      "I171.4" { ExternalVisible := 'False'} : Bool := FALSE;   // I171.4
      "I171.5" { ExternalVisible := 'False'} : Bool := FALSE;   // I171.5
      "I171.6" { ExternalVisible := 'False'} : Bool := FALSE;   // I171.6
      "I171.7" { ExternalVisible := 'False'} : Bool := FALSE;   // I171.7
      "I172.0" { ExternalVisible := 'False'} : Bool := FALSE;   // I172.0
      "I172.1" { ExternalVisible := 'False'} : Bool := FALSE;   // I172.1
      "I172.2" { ExternalVisible := 'False'} : Bool := FALSE;   // I172.2
      "I172.3" { ExternalVisible := 'False'} : Bool := FALSE;   // I172.3
      "I172.4" { ExternalVisible := 'False'} : Bool := FALSE;   // I172.4
      "I172.5" { ExternalVisible := 'False'} : Bool := FALSE;   // I172.5
      "I172.6" { ExternalVisible := 'False'} : Bool := FALSE;   // I172.6
      "I172.7" { ExternalVisible := 'False'} : Bool := FALSE;   // I172.7
      "I173.0" { ExternalVisible := 'False'} : Bool := FALSE;   // I173.0
      "I173.1" { ExternalVisible := 'False'} : Bool := FALSE;   // I173.1
      "I173.2" { ExternalVisible := 'False'} : Bool := FALSE;   // I173.2
      "I173.3" { ExternalVisible := 'False'} : Bool := FALSE;   // I173.3
      "I173.4" { ExternalVisible := 'False'} : Bool := FALSE;   // I173.4
      "I173.5" { ExternalVisible := 'False'} : Bool := FALSE;   // I173.5
      "I173.6" { ExternalVisible := 'False'} : Bool := FALSE;   // I173.6
      "I173.7" { ExternalVisible := 'False'} : Bool := FALSE;   // I173.7
      "I174.0" { ExternalVisible := 'False'} : Bool := FALSE;   // I174.0
      "I174.1" { ExternalVisible := 'False'} : Bool := FALSE;   // I174.1
      "I174.2" { ExternalVisible := 'False'} : Bool := FALSE;   // I174.2
      "I174.3" { ExternalVisible := 'False'} : Bool := FALSE;   // I174.3
      "I174.4" { ExternalVisible := 'False'} : Bool := FALSE;   // I174.4
      "I174.5" { ExternalVisible := 'False'} : Bool := FALSE;   // I174.5
      "I174.6" { ExternalVisible := 'False'} : Bool := FALSE;   // I174.6
      "I174.7" { ExternalVisible := 'False'} : Bool := FALSE;   // I174.7
      "I175.0" { ExternalVisible := 'False'} : Bool := FALSE;   // I175.0
      "I175.1" { ExternalVisible := 'False'} : Bool := FALSE;   // I175.1
      "I175.2" { ExternalVisible := 'False'} : Bool := FALSE;   // I175.2
      "I175.3" { ExternalVisible := 'False'} : Bool := FALSE;   // I175.3
      "I175.4" { ExternalVisible := 'False'} : Bool := FALSE;   // I175.4
      "I175.5" { ExternalVisible := 'False'} : Bool := FALSE;   // I175.5
      "I175.6" { ExternalVisible := 'False'} : Bool := FALSE;   // I175.6
      "I175.7" { ExternalVisible := 'False'} : Bool := FALSE;   // I175.7
      "I176.0" { ExternalVisible := 'False'} : Bool := FALSE;   // I176.0
      "I176.1" { ExternalVisible := 'False'} : Bool := FALSE;   // I176.1
      "I176.2" { ExternalVisible := 'False'} : Bool := FALSE;   // I176.2
      "I176.3" { ExternalVisible := 'False'} : Bool := FALSE;   // I176.3
      "I176.4" { ExternalVisible := 'False'} : Bool := FALSE;   // I176.4
      "I176.5" { ExternalVisible := 'False'} : Bool := FALSE;   // I176.5
      "I176.6" { ExternalVisible := 'False'} : Bool := FALSE;   // I176.6
      "I176.7" { ExternalVisible := 'False'} : Bool := FALSE;   // I176.7
      "I177.0" { ExternalVisible := 'False'} : Bool := FALSE;   // I177.0
      "I177.1" { ExternalVisible := 'False'} : Bool := FALSE;   // I177.1
      "I177.2" { ExternalVisible := 'False'} : Bool := FALSE;   // I177.2
      "I177.3" { ExternalVisible := 'False'} : Bool := FALSE;   // I177.3
      "I177.4" { ExternalVisible := 'False'} : Bool := FALSE;   // I177.4
      "I177.5" { ExternalVisible := 'False'} : Bool := FALSE;   // I177.5
      "I177.6" { ExternalVisible := 'False'} : Bool := FALSE;   // I177.6
      "I177.7" { ExternalVisible := 'False'} : Bool := FALSE;   // I177.7
      "I178.0" { ExternalVisible := 'False'} : Bool := FALSE;   // I178.0
      "I178.1" { ExternalVisible := 'False'} : Bool := FALSE;   // I178.1
      "I178.2" { ExternalVisible := 'False'} : Bool := FALSE;   // I178.2
      "I178.3" { ExternalVisible := 'False'} : Bool := FALSE;   // I178.3
      "I178.4" { ExternalVisible := 'False'} : Bool := FALSE;   // I178.4
      "I178.5" { ExternalVisible := 'False'} : Bool := FALSE;   // I178.5
      "I178.6" { ExternalVisible := 'False'} : Bool := FALSE;   // I178.6
      "I178.7" { ExternalVisible := 'False'} : Bool := FALSE;   // I178.7
      "I179.0" { ExternalVisible := 'False'} : Bool := FALSE;   // I179.0
      "I179.1" { ExternalVisible := 'False'} : Bool := FALSE;   // I179.1
      "I179.2" { ExternalVisible := 'False'} : Bool := FALSE;   // I179.2
      "I179.3" { ExternalVisible := 'False'} : Bool := FALSE;   // I179.3
      "I179.4" { ExternalVisible := 'False'} : Bool := FALSE;   // I179.4
      "I179.5" { ExternalVisible := 'False'} : Bool := FALSE;   // I179.5
      "I179.6" { ExternalVisible := 'False'} : Bool := FALSE;   // I179.6
      "I179.7" { ExternalVisible := 'False'} : Bool := FALSE;   // I179.7
      "I180.0" { ExternalVisible := 'False'} : Bool := FALSE;   // I180.0
      "I180.1" { ExternalVisible := 'False'} : Bool := FALSE;   // I180.1
      "I180.2" { ExternalVisible := 'False'} : Bool := FALSE;   // I180.2
      "I180.3" { ExternalVisible := 'False'} : Bool := FALSE;   // I180.3
      "I180.4" { ExternalVisible := 'False'} : Bool := FALSE;   // I180.4
      "I180.5" { ExternalVisible := 'False'} : Bool := FALSE;   // I180.5
      "I180.6" { ExternalVisible := 'False'} : Bool := FALSE;   // I180.6
      "I180.7" { ExternalVisible := 'False'} : Bool := FALSE;   // I180.7
      "I181.0" { ExternalVisible := 'False'} : Bool := FALSE;   // I181.0
      "I181.1" { ExternalVisible := 'False'} : Bool := FALSE;   // I181.1
      "I181.2" { ExternalVisible := 'False'} : Bool := FALSE;   // I181.2
      "I181.3" { ExternalVisible := 'False'} : Bool := FALSE;   // I181.3
      "I181.4" { ExternalVisible := 'False'} : Bool := FALSE;   // I181.4
      "I181.5" { ExternalVisible := 'False'} : Bool := FALSE;   // I181.5
      "I181.6" { ExternalVisible := 'False'} : Bool := FALSE;   // I181.6
      "I181.7" { ExternalVisible := 'False'} : Bool := FALSE;   // I181.7
      "I182.0" { ExternalVisible := 'False'} : Bool := FALSE;   // I182.0
      "I182.1" { ExternalVisible := 'False'} : Bool := FALSE;   // I182.1
      "I182.2" { ExternalVisible := 'False'} : Bool := FALSE;   // I182.2
      "I182.3" { ExternalVisible := 'False'} : Bool := FALSE;   // I182.3
      "I182.4" { ExternalVisible := 'False'} : Bool := FALSE;   // I182.4
      "I182.5" { ExternalVisible := 'False'} : Bool := FALSE;   // I182.5
      "I182.6" { ExternalVisible := 'False'} : Bool := FALSE;   // I182.6
      "I182.7" { ExternalVisible := 'False'} : Bool := FALSE;   // I182.7
      "I183.0" { ExternalVisible := 'False'} : Bool := FALSE;   // I183.0
      "I183.1" { ExternalVisible := 'False'} : Bool := FALSE;   // I183.1
      "I183.2" { ExternalVisible := 'False'} : Bool := FALSE;   // I183.2
      "I183.3" { ExternalVisible := 'False'} : Bool := FALSE;   // I183.3
      "I183.4" { ExternalVisible := 'False'} : Bool := FALSE;   // I183.4
      "I183.5" { ExternalVisible := 'False'} : Bool := FALSE;   // I183.5
      "I183.6" { ExternalVisible := 'False'} : Bool := FALSE;   // I183.6
      "I183.7" { ExternalVisible := 'False'} : Bool := FALSE;   // I183.7
      "I184.0" { ExternalVisible := 'False'} : Bool := FALSE;   // I184.0
      "I184.1" { ExternalVisible := 'False'} : Bool := FALSE;   // I184.1
      "I184.2" { ExternalVisible := 'False'} : Bool := FALSE;   // I184.2
      "I184.3" { ExternalVisible := 'False'} : Bool := FALSE;   // I184.3
      "I184.4" { ExternalVisible := 'False'} : Bool := FALSE;   // I184.4
      "I184.5" { ExternalVisible := 'False'} : Bool := FALSE;   // I184.5
      "I184.6" { ExternalVisible := 'False'} : Bool := FALSE;   // I184.6
      "I184.7" { ExternalVisible := 'False'} : Bool := FALSE;   // I184.7
      "I185.0" { ExternalVisible := 'False'} : Bool := FALSE;   // I185.0
      "I185.1" { ExternalVisible := 'False'} : Bool := FALSE;   // I185.1
      "I185.2" { ExternalVisible := 'False'} : Bool := FALSE;   // I185.2
      "I185.3" { ExternalVisible := 'False'} : Bool := FALSE;   // I185.3
      "I185.4" { ExternalVisible := 'False'} : Bool := FALSE;   // I185.4
      "I185.5" { ExternalVisible := 'False'} : Bool := FALSE;   // I185.5
      "I185.6" { ExternalVisible := 'False'} : Bool := FALSE;   // I185.6
      "I185.7" { ExternalVisible := 'False'} : Bool := FALSE;   // I185.7
      "I186.0" { ExternalVisible := 'False'} : Bool := FALSE;   // I186.0
      "I186.1" { ExternalVisible := 'False'} : Bool := FALSE;   // I186.1
      "I186.2" { ExternalVisible := 'False'} : Bool := FALSE;   // I186.2
      "I186.3" { ExternalVisible := 'False'} : Bool := FALSE;   // I186.3
      "I186.4" { ExternalVisible := 'False'} : Bool := FALSE;   // I186.4
      "I186.5" { ExternalVisible := 'False'} : Bool := FALSE;   // I186.5
      "I186.6" { ExternalVisible := 'False'} : Bool := FALSE;   // I186.6
      "I186.7" { ExternalVisible := 'False'} : Bool := FALSE;   // I186.7
      "I187.0" { ExternalVisible := 'False'} : Bool := FALSE;   // I187.0
      "I187.1" { ExternalVisible := 'False'} : Bool := FALSE;   // I187.1
      "I187.2" { ExternalVisible := 'False'} : Bool := FALSE;   // I187.2
      "I187.3" { ExternalVisible := 'False'} : Bool := FALSE;   // I187.3
      "I187.4" { ExternalVisible := 'False'} : Bool := FALSE;   // I187.4
      "I187.5" { ExternalVisible := 'False'} : Bool := FALSE;   // I187.5
      "I187.6" { ExternalVisible := 'False'} : Bool := FALSE;   // I187.6
      "I187.7" { ExternalVisible := 'False'} : Bool := FALSE;   // I187.7
      "I188.0" { ExternalVisible := 'False'} : Bool := FALSE;   // I188.0
      "I188.1" { ExternalVisible := 'False'} : Bool := FALSE;   // I188.1
      "I188.2" { ExternalVisible := 'False'} : Bool := FALSE;   // I188.2
      "I188.3" { ExternalVisible := 'False'} : Bool := FALSE;   // I188.3
      "I188.4" { ExternalVisible := 'False'} : Bool := FALSE;   // I188.4
      "I188.5" { ExternalVisible := 'False'} : Bool := FALSE;   // I188.5
      "I188.6" { ExternalVisible := 'False'} : Bool := FALSE;   // I188.6
      "I188.7" { ExternalVisible := 'False'} : Bool := FALSE;   // I188.7
      "I189.0" { ExternalVisible := 'False'} : Bool := FALSE;   // I189.0
      "I189.1" { ExternalVisible := 'False'} : Bool := FALSE;   // I189.1
      "I189.2" { ExternalVisible := 'False'} : Bool := FALSE;   // I189.2
      "I189.3" { ExternalVisible := 'False'} : Bool := FALSE;   // I189.3
      "I189.4" { ExternalVisible := 'False'} : Bool := FALSE;   // I189.4
      "I189.5" { ExternalVisible := 'False'} : Bool := FALSE;   // I189.5
      "I189.6" { ExternalVisible := 'False'} : Bool := FALSE;   // I189.6
      "I189.7" { ExternalVisible := 'False'} : Bool := FALSE;   // I189.7
      "I190.0" { ExternalVisible := 'False'} : Bool := FALSE;   // I190.0
      "I190.1" { ExternalVisible := 'False'} : Bool := FALSE;   // I190.1
      "I190.2" { ExternalVisible := 'False'} : Bool := FALSE;   // I190.2
      "I190.3" { ExternalVisible := 'False'} : Bool := FALSE;   // I190.3
      "I190.4" { ExternalVisible := 'False'} : Bool := FALSE;   // I190.4
      "I190.5" { ExternalVisible := 'False'} : Bool := FALSE;   // I190.5
      "I190.6" { ExternalVisible := 'False'} : Bool := FALSE;   // I190.6
      "I190.7" { ExternalVisible := 'False'} : Bool := FALSE;   // I190.7
      "I191.0" { ExternalVisible := 'False'} : Bool := FALSE;   // I191.0
      "I191.1" { ExternalVisible := 'False'} : Bool := FALSE;   // I191.1
      "I191.2" { ExternalVisible := 'False'} : Bool := FALSE;   // I191.2
      "I191.3" { ExternalVisible := 'False'} : Bool := FALSE;   // I191.3
      "I191.4" { ExternalVisible := 'False'} : Bool := FALSE;   // I191.4
      "I191.5" { ExternalVisible := 'False'} : Bool := FALSE;   // I191.5
      "I191.6" { ExternalVisible := 'False'} : Bool := FALSE;   // I191.6
      "I191.7" { ExternalVisible := 'False'} : Bool := FALSE;   // I191.7
      "I192.0" { ExternalVisible := 'False'} : Bool := FALSE;   // I192.0
      "I192.1" { ExternalVisible := 'False'} : Bool := FALSE;   // I192.1
      "I192.2" { ExternalVisible := 'False'} : Bool := FALSE;   // I192.2
      "I192.3" { ExternalVisible := 'False'} : Bool := FALSE;   // I192.3
      "I192.4" { ExternalVisible := 'False'} : Bool := FALSE;   // I192.4
      "I192.5" { ExternalVisible := 'False'} : Bool := FALSE;   // I192.5
      "I192.6" { ExternalVisible := 'False'} : Bool := FALSE;   // I192.6
      "I192.7" { ExternalVisible := 'False'} : Bool := FALSE;   // I192.7
      "I193.0" { ExternalVisible := 'False'} : Bool := FALSE;   // I193.0
      "I193.1" { ExternalVisible := 'False'} : Bool := FALSE;   // I193.1
      "I193.2" { ExternalVisible := 'False'} : Bool := FALSE;   // I193.2
      "I193.3" { ExternalVisible := 'False'} : Bool := FALSE;   // I193.3
      "I193.4" { ExternalVisible := 'False'} : Bool := FALSE;   // I193.4
      "I193.5" { ExternalVisible := 'False'} : Bool := FALSE;   // I193.5
      "I193.6" { ExternalVisible := 'False'} : Bool := FALSE;   // I193.6
      "I193.7" { ExternalVisible := 'False'} : Bool := FALSE;   // I193.7
      "I194.0" { ExternalVisible := 'False'} : Bool := FALSE;   // I194.0
      "I194.1" { ExternalVisible := 'False'} : Bool := FALSE;   // I194.1
      "I194.2" { ExternalVisible := 'False'} : Bool := FALSE;   // I194.2
      "I194.3" { ExternalVisible := 'False'} : Bool := FALSE;   // I194.3
      "I194.4" { ExternalVisible := 'False'} : Bool := FALSE;   // I194.4
      "I194.5" { ExternalVisible := 'False'} : Bool := FALSE;   // I194.5
      "I194.6" { ExternalVisible := 'False'} : Bool := FALSE;   // I194.6
      "I194.7" { ExternalVisible := 'False'} : Bool := FALSE;   // I194.7
      "I195.0" { ExternalVisible := 'False'} : Bool := FALSE;   // I195.0
      "I195.1" { ExternalVisible := 'False'} : Bool := FALSE;   // I195.1
      "I195.2" { ExternalVisible := 'False'} : Bool := FALSE;   // I195.2
      "I195.3" { ExternalVisible := 'False'} : Bool := FALSE;   // I195.3
      "I195.4" { ExternalVisible := 'False'} : Bool := FALSE;   // I195.4
      "I195.5" { ExternalVisible := 'False'} : Bool := FALSE;   // I195.5
      "I195.6" { ExternalVisible := 'False'} : Bool := FALSE;   // I195.6
      "I195.7" { ExternalVisible := 'False'} : Bool := FALSE;   // I195.7
      "I196.0" { ExternalVisible := 'False'} : Bool := FALSE;   // I196.0
      "I196.1" { ExternalVisible := 'False'} : Bool := FALSE;   // I196.1
      "I196.2" { ExternalVisible := 'False'} : Bool := FALSE;   // I196.2
      "I196.3" { ExternalVisible := 'False'} : Bool := FALSE;   // I196.3
      "I196.4" { ExternalVisible := 'False'} : Bool := FALSE;   // I196.4
      "I196.5" { ExternalVisible := 'False'} : Bool := FALSE;   // I196.5
      "I196.6" { ExternalVisible := 'False'} : Bool := FALSE;   // I196.6
      "I196.7" { ExternalVisible := 'False'} : Bool := FALSE;   // I196.7
      "I197.0" { ExternalVisible := 'False'} : Bool := FALSE;   // I197.0
      "I197.1" { ExternalVisible := 'False'} : Bool := FALSE;   // I197.1
      "I197.2" { ExternalVisible := 'False'} : Bool := FALSE;   // I197.2
      "I197.3" { ExternalVisible := 'False'} : Bool := FALSE;   // I197.3
      "I197.4" { ExternalVisible := 'False'} : Bool := FALSE;   // I197.4
      "I197.5" { ExternalVisible := 'False'} : Bool := FALSE;   // I197.5
      "I197.6" { ExternalVisible := 'False'} : Bool := FALSE;   // I197.6
      "I197.7" { ExternalVisible := 'False'} : Bool := FALSE;   // I197.7
      "I198.0" { ExternalVisible := 'False'} : Bool := FALSE;   // I198.0
      "I198.1" { ExternalVisible := 'False'} : Bool := FALSE;   // I198.1
      "I198.2" { ExternalVisible := 'False'} : Bool := FALSE;   // I198.2
      "I198.3" { ExternalVisible := 'False'} : Bool := FALSE;   // I198.3
      "I198.4" { ExternalVisible := 'False'} : Bool := FALSE;   // I198.4
      "I198.5" { ExternalVisible := 'False'} : Bool := FALSE;   // I198.5
      "I198.6" { ExternalVisible := 'False'} : Bool := FALSE;   // I198.6
      "I198.7" { ExternalVisible := 'False'} : Bool := FALSE;   // I198.7
      "I199.0" { ExternalVisible := 'False'} : Bool := FALSE;   // I199.0
      "I199.1" { ExternalVisible := 'False'} : Bool := FALSE;   // I199.1
      "I199.2" { ExternalVisible := 'False'} : Bool := FALSE;   // I199.2
      "I199.3" { ExternalVisible := 'False'} : Bool := FALSE;   // I199.3
      "I199.4" { ExternalVisible := 'False'} : Bool := FALSE;   // I199.4
      "I199.5" { ExternalVisible := 'False'} : Bool := FALSE;   // I199.5
      "I199.6" { ExternalVisible := 'False'} : Bool := FALSE;   // I199.6
      "I199.7" { ExternalVisible := 'False'} : Bool := FALSE;   // I199.7
      "I200.0" { ExternalVisible := 'False'} : Bool := FALSE;   // I200.0
      "I200.1" { ExternalVisible := 'False'} : Bool := FALSE;   // I200.1
      "I200.2" { ExternalVisible := 'False'} : Bool := FALSE;   // I200.2
      "I200.3" { ExternalVisible := 'False'} : Bool := FALSE;   // I200.3
      "I200.4" { ExternalVisible := 'False'} : Bool := FALSE;   // I200.4
      "I200.5" { ExternalVisible := 'False'} : Bool := FALSE;   // I200.5
      "I200.6" { ExternalVisible := 'False'} : Bool := FALSE;   // I200.6
      "I200.7" { ExternalVisible := 'False'} : Bool := FALSE;   // I200.7
      "I201.0" { ExternalVisible := 'False'} : Bool := FALSE;   // I201.0
      "I201.1" { ExternalVisible := 'False'} : Bool := FALSE;   // I201.1
      "I201.2" { ExternalVisible := 'False'} : Bool := FALSE;   // I201.2
      "I201.3" { ExternalVisible := 'False'} : Bool := FALSE;   // I201.3
      "I201.4" { ExternalVisible := 'False'} : Bool := FALSE;   // I201.4
      "I201.5" { ExternalVisible := 'False'} : Bool := FALSE;   // I201.5
      "I201.6" { ExternalVisible := 'False'} : Bool := FALSE;   // I201.6
      "I201.7" { ExternalVisible := 'False'} : Bool := FALSE;   // I201.7
      "I202.0" { ExternalVisible := 'False'} : Bool := FALSE;   // I202.0
      "I202.1" { ExternalVisible := 'False'} : Bool := FALSE;   // I202.1
      "I202.2" { ExternalVisible := 'False'} : Bool := FALSE;   // I202.2
      "I202.3" { ExternalVisible := 'False'} : Bool := FALSE;   // I202.3
      "I202.4" { ExternalVisible := 'False'} : Bool := FALSE;   // I202.4
      "I202.5" { ExternalVisible := 'False'} : Bool := FALSE;   // I202.5
      "I202.6" { ExternalVisible := 'False'} : Bool := FALSE;   // I202.6
      "I202.7" { ExternalVisible := 'False'} : Bool := FALSE;   // I202.7
      "I203.0" { ExternalVisible := 'False'} : Bool := FALSE;   // I203.0
      "I203.1" { ExternalVisible := 'False'} : Bool := FALSE;   // I203.1
      "I203.2" { ExternalVisible := 'False'} : Bool := FALSE;   // I203.2
      "I203.3" { ExternalVisible := 'False'} : Bool := FALSE;   // I203.3
      "I203.4" { ExternalVisible := 'False'} : Bool := FALSE;   // I203.4
      "I203.5" { ExternalVisible := 'False'} : Bool := FALSE;   // I203.5
      "I203.6" { ExternalVisible := 'False'} : Bool := FALSE;   // I203.6
      "I203.7" { ExternalVisible := 'False'} : Bool := FALSE;   // I203.7
      "I204.0" { ExternalVisible := 'False'} : Bool := FALSE;   // I204.0
      "I204.1" { ExternalVisible := 'False'} : Bool := FALSE;   // I204.1
      "I204.2" { ExternalVisible := 'False'} : Bool := FALSE;   // I204.2
      "I204.3" { ExternalVisible := 'False'} : Bool := FALSE;   // I204.3
      "I204.4" { ExternalVisible := 'False'} : Bool := FALSE;   // I204.4
      "I204.5" { ExternalVisible := 'False'} : Bool := FALSE;   // I204.5
      "I204.6" { ExternalVisible := 'False'} : Bool := FALSE;   // I204.6
      "I204.7" { ExternalVisible := 'False'} : Bool := FALSE;   // I204.7
      "I205.0" { ExternalVisible := 'False'} : Bool := FALSE;   // I205.0
      "I205.1" { ExternalVisible := 'False'} : Bool := FALSE;   // I205.1
      "I205.2" { ExternalVisible := 'False'} : Bool := FALSE;   // I205.2
      "I205.3" { ExternalVisible := 'False'} : Bool := FALSE;   // I205.3
      "I205.4" { ExternalVisible := 'False'} : Bool := FALSE;   // I205.4
      "I205.5" { ExternalVisible := 'False'} : Bool := FALSE;   // I205.5
      "I205.6" { ExternalVisible := 'False'} : Bool := FALSE;   // I205.6
      "I205.7" { ExternalVisible := 'False'} : Bool := FALSE;   // I205.7
      "I206.0" { ExternalVisible := 'False'} : Bool := FALSE;   // I206.0
      "I206.1" { ExternalVisible := 'False'} : Bool := FALSE;   // I206.1
      "I206.2" { ExternalVisible := 'False'} : Bool := FALSE;   // I206.2
      "I206.3" { ExternalVisible := 'False'} : Bool := FALSE;   // I206.3
      "I206.4" { ExternalVisible := 'False'} : Bool := FALSE;   // I206.4
      "I206.5" { ExternalVisible := 'False'} : Bool := FALSE;   // I206.5
      "I206.6" { ExternalVisible := 'False'} : Bool := FALSE;   // I206.6
      "I206.7" { ExternalVisible := 'False'} : Bool := FALSE;   // I206.7
      "I207.0" { ExternalVisible := 'False'} : Bool := FALSE;   // I207.0
      "I207.1" { ExternalVisible := 'False'} : Bool := FALSE;   // I207.1
      "I207.2" { ExternalVisible := 'False'} : Bool := FALSE;   // I207.2
      "I207.3" { ExternalVisible := 'False'} : Bool := FALSE;   // I207.3
      "I207.4" { ExternalVisible := 'False'} : Bool := FALSE;   // I207.4
      "I207.5" { ExternalVisible := 'False'} : Bool := FALSE;   // I207.5
      "I207.6" { ExternalVisible := 'False'} : Bool := FALSE;   // I207.6
      "I207.7" { ExternalVisible := 'False'} : Bool := FALSE;   // I207.7
      "I208.0" { ExternalVisible := 'False'} : Bool := FALSE;   // I208.0
      "I208.1" { ExternalVisible := 'False'} : Bool := FALSE;   // I208.1
      "I208.2" { ExternalVisible := 'False'} : Bool := FALSE;   // I208.2
      "I208.3" { ExternalVisible := 'False'} : Bool := FALSE;   // I208.3
      "I208.4" { ExternalVisible := 'False'} : Bool := FALSE;   // I208.4
      "I208.5" { ExternalVisible := 'False'} : Bool := FALSE;   // I208.5
      "I208.6" { ExternalVisible := 'False'} : Bool := FALSE;   // I208.6
      "I208.7" { ExternalVisible := 'False'} : Bool := FALSE;   // I208.7
      "I209.0" { ExternalVisible := 'False'} : Bool := FALSE;   // I209.0
      "I209.1" { ExternalVisible := 'False'} : Bool := FALSE;   // I209.1
      "I209.2" { ExternalVisible := 'False'} : Bool := FALSE;   // I209.2
      "I209.3" { ExternalVisible := 'False'} : Bool := FALSE;   // I209.3
      "I209.4" { ExternalVisible := 'False'} : Bool := FALSE;   // I209.4
      "I209.5" { ExternalVisible := 'False'} : Bool := FALSE;   // I209.5
      "I209.6" { ExternalVisible := 'False'} : Bool := FALSE;   // I209.6
      "I209.7" { ExternalVisible := 'False'} : Bool := FALSE;   // I209.7
      "I210.0" { ExternalVisible := 'False'} : Bool := FALSE;   // I210.0
      "I210.1" { ExternalVisible := 'False'} : Bool := FALSE;   // I210.1
      "I210.2" { ExternalVisible := 'False'} : Bool := FALSE;   // I210.2
      "I210.3" { ExternalVisible := 'False'} : Bool := FALSE;   // I210.3
      "I210.4" { ExternalVisible := 'False'} : Bool := FALSE;   // I210.4
      "I210.5" { ExternalVisible := 'False'} : Bool := FALSE;   // I210.5
      "I210.6" { ExternalVisible := 'False'} : Bool := FALSE;   // I210.6
      "I210.7" { ExternalVisible := 'False'} : Bool := FALSE;   // I210.7
      "I211.0" { ExternalVisible := 'False'} : Bool := FALSE;   // I211.0
      "I211.1" { ExternalVisible := 'False'} : Bool := FALSE;   // I211.1
      "I211.2" { ExternalVisible := 'False'} : Bool := FALSE;   // I211.2
      "I211.3" { ExternalVisible := 'False'} : Bool := FALSE;   // I211.3
      "I211.4" { ExternalVisible := 'False'} : Bool := FALSE;   // I211.4
      "I211.5" { ExternalVisible := 'False'} : Bool := FALSE;   // I211.5
      "I211.6" { ExternalVisible := 'False'} : Bool := FALSE;   // I211.6
      "I211.7" { ExternalVisible := 'False'} : Bool := FALSE;   // I211.7
      "I212.0" { ExternalVisible := 'False'} : Bool := FALSE;   // I212.0
      "I212.1" { ExternalVisible := 'False'} : Bool := FALSE;   // I212.1
      "I212.2" { ExternalVisible := 'False'} : Bool := FALSE;   // I212.2
      "I212.3" { ExternalVisible := 'False'} : Bool := FALSE;   // I212.3
      "I212.4" { ExternalVisible := 'False'} : Bool := FALSE;   // I212.4
      "I212.5" { ExternalVisible := 'False'} : Bool := FALSE;   // I212.5
      "I212.6" { ExternalVisible := 'False'} : Bool := FALSE;   // I212.6
      "I212.7" { ExternalVisible := 'False'} : Bool := FALSE;   // I212.7
      "I213.0" { ExternalVisible := 'False'} : Bool := FALSE;   // I213.0
      "I213.1" { ExternalVisible := 'False'} : Bool := FALSE;   // I213.1
      "I213.2" { ExternalVisible := 'False'} : Bool := FALSE;   // I213.2
      "I213.3" { ExternalVisible := 'False'} : Bool := FALSE;   // I213.3
      "I213.4" { ExternalVisible := 'False'} : Bool := FALSE;   // I213.4
      "I213.5" { ExternalVisible := 'False'} : Bool := FALSE;   // I213.5
      "I213.6" { ExternalVisible := 'False'} : Bool := FALSE;   // I213.6
      "I213.7" { ExternalVisible := 'False'} : Bool := FALSE;   // I213.7
      "I214.0" { ExternalVisible := 'False'} : Bool := FALSE;   // I214.0
      "I214.1" { ExternalVisible := 'False'} : Bool := FALSE;   // I214.1
      "I214.2" { ExternalVisible := 'False'} : Bool := FALSE;   // I214.2
      "I214.3" { ExternalVisible := 'False'} : Bool := FALSE;   // I214.3
      "I214.4" { ExternalVisible := 'False'} : Bool := FALSE;   // I214.4
      "I214.5" { ExternalVisible := 'False'} : Bool := FALSE;   // I214.5
      "I214.6" { ExternalVisible := 'False'} : Bool := FALSE;   // I214.6
      "I214.7" { ExternalVisible := 'False'} : Bool := FALSE;   // I214.7
      "I215.0" { ExternalVisible := 'False'} : Bool := FALSE;   // I215.0
      "I215.1" { ExternalVisible := 'False'} : Bool := FALSE;   // I215.1
      "I215.2" { ExternalVisible := 'False'} : Bool := FALSE;   // I215.2
      "I215.3" { ExternalVisible := 'False'} : Bool := FALSE;   // I215.3
      "I215.4" { ExternalVisible := 'False'} : Bool := FALSE;   // I215.4
      "I215.5" { ExternalVisible := 'False'} : Bool := FALSE;   // I215.5
      "I215.6" { ExternalVisible := 'False'} : Bool := FALSE;   // I215.6
      "I215.7" { ExternalVisible := 'False'} : Bool := FALSE;   // I215.7
      "I216.0" { ExternalVisible := 'False'} : Bool := FALSE;   // I216.0
      "I216.1" { ExternalVisible := 'False'} : Bool := FALSE;   // I216.1
      "I216.2" { ExternalVisible := 'False'} : Bool := FALSE;   // I216.2
      "I216.3" { ExternalVisible := 'False'} : Bool := FALSE;   // I216.3
      "I216.4" { ExternalVisible := 'False'} : Bool := FALSE;   // I216.4
      "I216.5" { ExternalVisible := 'False'} : Bool := FALSE;   // I216.5
      "I216.6" { ExternalVisible := 'False'} : Bool := FALSE;   // I216.6
      "I216.7" { ExternalVisible := 'False'} : Bool := FALSE;   // I216.7
      "I217.0" { ExternalVisible := 'False'} : Bool := FALSE;   // I217.0
      "I217.1" { ExternalVisible := 'False'} : Bool := FALSE;   // I217.1
      "I217.2" { ExternalVisible := 'False'} : Bool := FALSE;   // I217.2
      "I217.3" { ExternalVisible := 'False'} : Bool := FALSE;   // I217.3
      "I217.4" { ExternalVisible := 'False'} : Bool := FALSE;   // I217.4
      "I217.5" { ExternalVisible := 'False'} : Bool := FALSE;   // I217.5
      "I217.6" { ExternalVisible := 'False'} : Bool := FALSE;   // I217.6
      "I217.7" { ExternalVisible := 'False'} : Bool := FALSE;   // I217.7
      "I218.0" { ExternalVisible := 'False'} : Bool := FALSE;   // I218.0
      "I218.1" { ExternalVisible := 'False'} : Bool := FALSE;   // I218.1
      "I218.2" { ExternalVisible := 'False'} : Bool := FALSE;   // I218.2
      "I218.3" { ExternalVisible := 'False'} : Bool := FALSE;   // I218.3
      "I218.4" { ExternalVisible := 'False'} : Bool := FALSE;   // I218.4
      "I218.5" { ExternalVisible := 'False'} : Bool := FALSE;   // I218.5
      "I218.6" { ExternalVisible := 'False'} : Bool := FALSE;   // I218.6
      "I218.7" { ExternalVisible := 'False'} : Bool := FALSE;   // I218.7
      "I219.0" { ExternalVisible := 'False'} : Bool := FALSE;   // I219.0
      "I219.1" { ExternalVisible := 'False'} : Bool := FALSE;   // I219.1
      "I219.2" { ExternalVisible := 'False'} : Bool := FALSE;   // I219.2
      "I219.3" { ExternalVisible := 'False'} : Bool := FALSE;   // I219.3
      "I219.4" { ExternalVisible := 'False'} : Bool := FALSE;   // I219.4
      "I219.5" { ExternalVisible := 'False'} : Bool := FALSE;   // I219.5
      "I219.6" { ExternalVisible := 'False'} : Bool := FALSE;   // I219.6
      "I219.7" { ExternalVisible := 'False'} : Bool := FALSE;   // I219.7
      "I220.0" { ExternalVisible := 'False'} : Bool := FALSE;   // I220.0
      "I220.1" { ExternalVisible := 'False'} : Bool := FALSE;   // I220.1
      "I220.2" { ExternalVisible := 'False'} : Bool := FALSE;   // I220.2
      "I220.3" { ExternalVisible := 'False'} : Bool := FALSE;   // I220.3
      "I220.4" { ExternalVisible := 'False'} : Bool := FALSE;   // I220.4
      "I220.5" { ExternalVisible := 'False'} : Bool := FALSE;   // I220.5
      "I220.6" { ExternalVisible := 'False'} : Bool := FALSE;   // I220.6
      "I220.7" { ExternalVisible := 'False'} : Bool := FALSE;   // I220.7
      "I221.0" { ExternalVisible := 'False'} : Bool := FALSE;   // I221.0
      "I221.1" { ExternalVisible := 'False'} : Bool := FALSE;   // I221.1
      "I221.2" { ExternalVisible := 'False'} : Bool := FALSE;   // I221.2
      "I221.3" { ExternalVisible := 'False'} : Bool := FALSE;   // I221.3
      "I221.4" { ExternalVisible := 'False'} : Bool := FALSE;   // I221.4
      "I221.5" { ExternalVisible := 'False'} : Bool := FALSE;   // I221.5
      "I221.6" { ExternalVisible := 'False'} : Bool := FALSE;   // I221.6
      "I221.7" { ExternalVisible := 'False'} : Bool := FALSE;   // I221.7
      "I222.0" { ExternalVisible := 'False'} : Bool := FALSE;   // I222.0
      "I222.1" { ExternalVisible := 'False'} : Bool := FALSE;   // I222.1
      "I222.2" { ExternalVisible := 'False'} : Bool := FALSE;   // I222.2
      "I222.3" { ExternalVisible := 'False'} : Bool := FALSE;   // I222.3
      "I222.4" { ExternalVisible := 'False'} : Bool := FALSE;   // I222.4
      "I222.5" { ExternalVisible := 'False'} : Bool := FALSE;   // I222.5
      "I222.6" { ExternalVisible := 'False'} : Bool := FALSE;   // I222.6
      "I222.7" { ExternalVisible := 'False'} : Bool := FALSE;   // I222.7
      "I223.0" { ExternalVisible := 'False'} : Bool := FALSE;   // I223.0
      "I223.1" { ExternalVisible := 'False'} : Bool := FALSE;   // I223.1
      "I223.2" { ExternalVisible := 'False'} : Bool := FALSE;   // I223.2
      "I223.3" { ExternalVisible := 'False'} : Bool := FALSE;   // I223.3
      "I223.4" { ExternalVisible := 'False'} : Bool := FALSE;   // I223.4
      "I223.5" { ExternalVisible := 'False'} : Bool := FALSE;   // I223.5
      "I223.6" { ExternalVisible := 'False'} : Bool := FALSE;   // I223.6
      "I223.7" { ExternalVisible := 'False'} : Bool := FALSE;   // I223.7
      "I224.0" { ExternalVisible := 'False'} : Bool := FALSE;   // I224.0
      "I224.1" { ExternalVisible := 'False'} : Bool := FALSE;   // I224.1
      "I224.2" { ExternalVisible := 'False'} : Bool := FALSE;   // I224.2
      "I224.3" { ExternalVisible := 'False'} : Bool := FALSE;   // I224.3
      "I224.4" { ExternalVisible := 'False'} : Bool := FALSE;   // I224.4
      "I224.5" { ExternalVisible := 'False'} : Bool := FALSE;   // I224.5
      "I224.6" { ExternalVisible := 'False'} : Bool := FALSE;   // I224.6
      "I224.7" { ExternalVisible := 'False'} : Bool := FALSE;   // I224.7
      "I225.0" { ExternalVisible := 'False'} : Bool := FALSE;   // I225.0
      "I225.1" { ExternalVisible := 'False'} : Bool := FALSE;   // I225.1
      "I225.2" { ExternalVisible := 'False'} : Bool := FALSE;   // I225.2
      "I225.3" { ExternalVisible := 'False'} : Bool := FALSE;   // I225.3
      "I225.4" { ExternalVisible := 'False'} : Bool := FALSE;   // I225.4
      "I225.5" { ExternalVisible := 'False'} : Bool := FALSE;   // I225.5
      "I225.6" { ExternalVisible := 'False'} : Bool := FALSE;   // I225.6
      "I225.7" { ExternalVisible := 'False'} : Bool := FALSE;   // I225.7
      "I226.0" { ExternalVisible := 'False'} : Bool := FALSE;   // I226.0
      "I226.1" { ExternalVisible := 'False'} : Bool := FALSE;   // I226.1
      "I226.2" { ExternalVisible := 'False'} : Bool := FALSE;   // I226.2
      "I226.3" { ExternalVisible := 'False'} : Bool := FALSE;   // I226.3
      "I226.4" { ExternalVisible := 'False'} : Bool := FALSE;   // I226.4
      "I226.5" { ExternalVisible := 'False'} : Bool := FALSE;   // I226.5
      "I226.6" { ExternalVisible := 'False'} : Bool := FALSE;   // I226.6
      "I226.7" { ExternalVisible := 'False'} : Bool := FALSE;   // I226.7
      "I227.0" { ExternalVisible := 'False'} : Bool := FALSE;   // I227.0
      "I227.1" { ExternalVisible := 'False'} : Bool := FALSE;   // I227.1
      "I227.2" { ExternalVisible := 'False'} : Bool := FALSE;   // I227.2
      "I227.3" { ExternalVisible := 'False'} : Bool := FALSE;   // I227.3
      "I227.4" { ExternalVisible := 'False'} : Bool := FALSE;   // I227.4
      "I227.5" { ExternalVisible := 'False'} : Bool := FALSE;   // I227.5
      "I227.6" { ExternalVisible := 'False'} : Bool := FALSE;   // I227.6
      "I227.7" { ExternalVisible := 'False'} : Bool := FALSE;   // I227.7
      "I228.0" { ExternalVisible := 'False'} : Bool := FALSE;   // I228.0
      "I228.1" { ExternalVisible := 'False'} : Bool := FALSE;   // I228.1
      "I228.2" { ExternalVisible := 'False'} : Bool := FALSE;   // I228.2
      "I228.3" { ExternalVisible := 'False'} : Bool := FALSE;   // I228.3
      "I228.4" { ExternalVisible := 'False'} : Bool := FALSE;   // I228.4
      "I228.5" { ExternalVisible := 'False'} : Bool := FALSE;   // I228.5
      "I228.6" { ExternalVisible := 'False'} : Bool := FALSE;   // I228.6
      "I228.7" { ExternalVisible := 'False'} : Bool := FALSE;   // I228.7
      "I229.0" { ExternalVisible := 'False'} : Bool := FALSE;   // I229.0
      "I229.1" { ExternalVisible := 'False'} : Bool := FALSE;   // I229.1
      "I229.2" { ExternalVisible := 'False'} : Bool := FALSE;   // I229.2
      "I229.3" { ExternalVisible := 'False'} : Bool := FALSE;   // I229.3
      "I229.4" { ExternalVisible := 'False'} : Bool := FALSE;   // I229.4
      "I229.5" { ExternalVisible := 'False'} : Bool := FALSE;   // I229.5
      "I229.6" { ExternalVisible := 'False'} : Bool := FALSE;   // I229.6
      "I229.7" { ExternalVisible := 'False'} : Bool := FALSE;   // I229.7
      "I230.0" { ExternalVisible := 'False'} : Bool := FALSE;   // I230.0
      "I230.1" { ExternalVisible := 'False'} : Bool := FALSE;   // I230.1
      "I230.2" { ExternalVisible := 'False'} : Bool := FALSE;   // I230.2
      "I230.3" { ExternalVisible := 'False'} : Bool := FALSE;   // I230.3
      "I230.4" { ExternalVisible := 'False'} : Bool := FALSE;   // I230.4
      "I230.5" { ExternalVisible := 'False'} : Bool := FALSE;   // I230.5
      "I230.6" { ExternalVisible := 'False'} : Bool := FALSE;   // I230.6
      "I230.7" { ExternalVisible := 'False'} : Bool := FALSE;   // I230.7
      "I231.0" { ExternalVisible := 'False'} : Bool := FALSE;   // I231.0
      "I231.1" { ExternalVisible := 'False'} : Bool := FALSE;   // I231.1
      "I231.2" { ExternalVisible := 'False'} : Bool := FALSE;   // I231.2
      "I231.3" { ExternalVisible := 'False'} : Bool := FALSE;   // I231.3
      "I231.4" { ExternalVisible := 'False'} : Bool := FALSE;   // I231.4
      "I231.5" { ExternalVisible := 'False'} : Bool := FALSE;   // I231.5
      "I231.6" { ExternalVisible := 'False'} : Bool := FALSE;   // I231.6
      "I231.7" { ExternalVisible := 'False'} : Bool := FALSE;   // I231.7
      "I232.0" { ExternalVisible := 'False'} : Bool := FALSE;   // I232.0
      "I232.1" { ExternalVisible := 'False'} : Bool := FALSE;   // I232.1
      "I232.2" { ExternalVisible := 'False'} : Bool := FALSE;   // I232.2
      "I232.3" { ExternalVisible := 'False'} : Bool := FALSE;   // I232.3
      "I232.4" { ExternalVisible := 'False'} : Bool := FALSE;   // I232.4
      "I232.5" { ExternalVisible := 'False'} : Bool := FALSE;   // I232.5
      "I232.6" { ExternalVisible := 'False'} : Bool := FALSE;   // I232.6
      "I232.7" { ExternalVisible := 'False'} : Bool := FALSE;   // I232.7
      "I233.0" { ExternalVisible := 'False'} : Bool := FALSE;   // I233.0
      "I233.1" { ExternalVisible := 'False'} : Bool := FALSE;   // I233.1
      "I233.2" { ExternalVisible := 'False'} : Bool := FALSE;   // I233.2
      "I233.3" { ExternalVisible := 'False'} : Bool := FALSE;   // I233.3
      "I233.4" { ExternalVisible := 'False'} : Bool := FALSE;   // I233.4
      "I233.5" { ExternalVisible := 'False'} : Bool := FALSE;   // I233.5
      "I233.6" { ExternalVisible := 'False'} : Bool := FALSE;   // I233.6
      "I233.7" { ExternalVisible := 'False'} : Bool := FALSE;   // I233.7
      "I234.0" { ExternalVisible := 'False'} : Bool := FALSE;   // I234.0
      "I234.1" { ExternalVisible := 'False'} : Bool := FALSE;   // I234.1
      "I234.2" { ExternalVisible := 'False'} : Bool := FALSE;   // I234.2
      "I234.3" { ExternalVisible := 'False'} : Bool := FALSE;   // I234.3
      "I234.4" { ExternalVisible := 'False'} : Bool := FALSE;   // I234.4
      "I234.5" { ExternalVisible := 'False'} : Bool := FALSE;   // I234.5
      "I234.6" { ExternalVisible := 'False'} : Bool := FALSE;   // I234.6
      "I234.7" { ExternalVisible := 'False'} : Bool := FALSE;   // I234.7
      "I235.0" { ExternalVisible := 'False'} : Bool := FALSE;   // I235.0
      "I235.1" { ExternalVisible := 'False'} : Bool := FALSE;   // I235.1
      "I235.2" { ExternalVisible := 'False'} : Bool := FALSE;   // I235.2
      "I235.3" { ExternalVisible := 'False'} : Bool := FALSE;   // I235.3
      "I235.4" { ExternalVisible := 'False'} : Bool := FALSE;   // I235.4
      "I235.5" { ExternalVisible := 'False'} : Bool := FALSE;   // I235.5
      "I235.6" { ExternalVisible := 'False'} : Bool := FALSE;   // I235.6
      "I235.7" { ExternalVisible := 'False'} : Bool := FALSE;   // I235.7
      "I236.0" { ExternalVisible := 'False'} : Bool := FALSE;   // I236.0
      "I236.1" { ExternalVisible := 'False'} : Bool := FALSE;   // I236.1
      "I236.2" { ExternalVisible := 'False'} : Bool := FALSE;   // I236.2
      "I236.3" { ExternalVisible := 'False'} : Bool := FALSE;   // I236.3
      "I236.4" { ExternalVisible := 'False'} : Bool := FALSE;   // I236.4
      "I236.5" { ExternalVisible := 'False'} : Bool := FALSE;   // I236.5
      "I236.6" { ExternalVisible := 'False'} : Bool := FALSE;   // I236.6
      "I236.7" { ExternalVisible := 'False'} : Bool := FALSE;   // I236.7
      "I237.0" { ExternalVisible := 'False'} : Bool := FALSE;   // I237.0
      "I237.1" { ExternalVisible := 'False'} : Bool := FALSE;   // I237.1
      "I237.2" { ExternalVisible := 'False'} : Bool := FALSE;   // I237.2
      "I237.3" { ExternalVisible := 'False'} : Bool := FALSE;   // I237.3
      "I237.4" { ExternalVisible := 'False'} : Bool := FALSE;   // I237.4
      "I237.5" { ExternalVisible := 'False'} : Bool := FALSE;   // I237.5
      "I237.6" { ExternalVisible := 'False'} : Bool := FALSE;   // I237.6
      "I237.7" { ExternalVisible := 'False'} : Bool := FALSE;   // I237.7
      "I238.0" { ExternalVisible := 'False'} : Bool := FALSE;   // I238.0
      "I238.1" { ExternalVisible := 'False'} : Bool := FALSE;   // I238.1
      "I238.2" { ExternalVisible := 'False'} : Bool := FALSE;   // I238.2
      "I238.3" { ExternalVisible := 'False'} : Bool := FALSE;   // I238.3
      "I238.4" { ExternalVisible := 'False'} : Bool := FALSE;   // I238.4
      "I238.5" { ExternalVisible := 'False'} : Bool := FALSE;   // I238.5
      "I238.6" { ExternalVisible := 'False'} : Bool := FALSE;   // I238.6
      "I238.7" { ExternalVisible := 'False'} : Bool := FALSE;   // I238.7
      "I239.0" { ExternalVisible := 'False'} : Bool := FALSE;   // I239.0
      "I239.1" { ExternalVisible := 'False'} : Bool := FALSE;   // I239.1
      "I239.2" { ExternalVisible := 'False'} : Bool := FALSE;   // I239.2
      "I239.3" { ExternalVisible := 'False'} : Bool := FALSE;   // I239.3
      "I239.4" { ExternalVisible := 'False'} : Bool := FALSE;   // I239.4
      "I239.5" { ExternalVisible := 'False'} : Bool := FALSE;   // I239.5
      "I239.6" { ExternalVisible := 'False'} : Bool := FALSE;   // I239.6
      "I239.7" { ExternalVisible := 'False'} : Bool := FALSE;   // I239.7
      "I240.0" { ExternalVisible := 'False'} : Bool := FALSE;   // I240.0
      "I240.1" { ExternalVisible := 'False'} : Bool := FALSE;   // I240.1
      "I240.2" { ExternalVisible := 'False'} : Bool := FALSE;   // I240.2
      "I240.3" { ExternalVisible := 'False'} : Bool := FALSE;   // I240.3
      "I240.4" { ExternalVisible := 'False'} : Bool := FALSE;   // I240.4
      "I240.5" { ExternalVisible := 'False'} : Bool := FALSE;   // I240.5
      "I240.6" { ExternalVisible := 'False'} : Bool := FALSE;   // I240.6
      "I240.7" { ExternalVisible := 'False'} : Bool := FALSE;   // I240.7
      "I241.0" { ExternalVisible := 'False'} : Bool := FALSE;   // I241.0
      "I241.1" { ExternalVisible := 'False'} : Bool := FALSE;   // I241.1
      "I241.2" { ExternalVisible := 'False'} : Bool := FALSE;   // I241.2
      "I241.3" { ExternalVisible := 'False'} : Bool := FALSE;   // I241.3
      "I241.4" { ExternalVisible := 'False'} : Bool := FALSE;   // I241.4
      "I241.5" { ExternalVisible := 'False'} : Bool := FALSE;   // I241.5
      "I241.6" { ExternalVisible := 'False'} : Bool := FALSE;   // I241.6
      "I241.7" { ExternalVisible := 'False'} : Bool := FALSE;   // I241.7
      "I242.0" { ExternalVisible := 'False'} : Bool := FALSE;   // I242.0
      "I242.1" { ExternalVisible := 'False'} : Bool := FALSE;   // I242.1
      "I242.2" { ExternalVisible := 'False'} : Bool := FALSE;   // I242.2
      "I242.3" { ExternalVisible := 'False'} : Bool := FALSE;   // I242.3
      "I242.4" { ExternalVisible := 'False'} : Bool := FALSE;   // I242.4
      "I242.5" { ExternalVisible := 'False'} : Bool := FALSE;   // I242.5
      "I242.6" { ExternalVisible := 'False'} : Bool := FALSE;   // I242.6
      "I242.7" { ExternalVisible := 'False'} : Bool := FALSE;   // I242.7
      "I243.0" { ExternalVisible := 'False'} : Bool := FALSE;   // I243.0
      "I243.1" { ExternalVisible := 'False'} : Bool := FALSE;   // I243.1
      "I243.2" { ExternalVisible := 'False'} : Bool := FALSE;   // I243.2
      "I243.3" { ExternalVisible := 'False'} : Bool := FALSE;   // I243.3
      "I243.4" { ExternalVisible := 'False'} : Bool := FALSE;   // I243.4
      "I243.5" { ExternalVisible := 'False'} : Bool := FALSE;   // I243.5
      "I243.6" { ExternalVisible := 'False'} : Bool := FALSE;   // I243.6
      "I243.7" { ExternalVisible := 'False'} : Bool := FALSE;   // I243.7
      "I244.0" { ExternalVisible := 'False'} : Bool := FALSE;   // I244.0
      "I244.1" { ExternalVisible := 'False'} : Bool := FALSE;   // I244.1
      "I244.2" { ExternalVisible := 'False'} : Bool := FALSE;   // I244.2
      "I244.3" { ExternalVisible := 'False'} : Bool := FALSE;   // I244.3
      "I244.4" { ExternalVisible := 'False'} : Bool := FALSE;   // I244.4
      "I244.5" { ExternalVisible := 'False'} : Bool := FALSE;   // I244.5
      "I244.6" { ExternalVisible := 'False'} : Bool := FALSE;   // I244.6
      "I244.7" { ExternalVisible := 'False'} : Bool := FALSE;   // I244.7
      "I245.0" { ExternalVisible := 'False'} : Bool := FALSE;   // I245.0
      "I245.1" { ExternalVisible := 'False'} : Bool := FALSE;   // I245.1
      "I245.2" { ExternalVisible := 'False'} : Bool := FALSE;   // I245.2
      "I245.3" { ExternalVisible := 'False'} : Bool := FALSE;   // I245.3
      "I245.4" { ExternalVisible := 'False'} : Bool := FALSE;   // I245.4
      "I245.5" { ExternalVisible := 'False'} : Bool := FALSE;   // I245.5
      "I245.6" { ExternalVisible := 'False'} : Bool := FALSE;   // I245.6
      "I245.7" { ExternalVisible := 'False'} : Bool := FALSE;   // I245.7
      "I246.0" { ExternalVisible := 'False'} : Bool := FALSE;   // I246.0
      "I246.1" { ExternalVisible := 'False'} : Bool := FALSE;   // I246.1
      "I246.2" { ExternalVisible := 'False'} : Bool := FALSE;   // I246.2
      "I246.3" { ExternalVisible := 'False'} : Bool := FALSE;   // I246.3
      "I246.4" { ExternalVisible := 'False'} : Bool := FALSE;   // I246.4
      "I246.5" { ExternalVisible := 'False'} : Bool := FALSE;   // I246.5
      "I246.6" { ExternalVisible := 'False'} : Bool := FALSE;   // I246.6
      "I246.7" { ExternalVisible := 'False'} : Bool := FALSE;   // I246.7
      "I247.0" { ExternalVisible := 'False'} : Bool := FALSE;   // I247.0
      "I247.1" { ExternalVisible := 'False'} : Bool := FALSE;   // I247.1
      "I247.2" { ExternalVisible := 'False'} : Bool := FALSE;   // I247.2
      "I247.3" { ExternalVisible := 'False'} : Bool := FALSE;   // I247.3
      "I247.4" { ExternalVisible := 'False'} : Bool := FALSE;   // I247.4
      "I247.5" { ExternalVisible := 'False'} : Bool := FALSE;   // I247.5
      "I247.6" { ExternalVisible := 'False'} : Bool := FALSE;   // I247.6
      "I247.7" { ExternalVisible := 'False'} : Bool := FALSE;   // I247.7
      "I248.0" { ExternalVisible := 'False'} : Bool := FALSE;   // I248.0
      "I248.1" { ExternalVisible := 'False'} : Bool := FALSE;   // I248.1
      "I248.2" { ExternalVisible := 'False'} : Bool := FALSE;   // I248.2
      "I248.3" { ExternalVisible := 'False'} : Bool := FALSE;   // I248.3
      "I248.4" { ExternalVisible := 'False'} : Bool := FALSE;   // I248.4
      "I248.5" { ExternalVisible := 'False'} : Bool := FALSE;   // I248.5
      "I248.6" { ExternalVisible := 'False'} : Bool := FALSE;   // I248.6
      "I248.7" { ExternalVisible := 'False'} : Bool := FALSE;   // I248.7
      "I249.0" { ExternalVisible := 'False'} : Bool := FALSE;   // I249.0
      "I249.1" { ExternalVisible := 'False'} : Bool := FALSE;   // I249.1
      "I249.2" { ExternalVisible := 'False'} : Bool := FALSE;   // I249.2
      "I249.3" { ExternalVisible := 'False'} : Bool := FALSE;   // I249.3
      "I249.4" { ExternalVisible := 'False'} : Bool := FALSE;   // I249.4
      "I249.5" { ExternalVisible := 'False'} : Bool := FALSE;   // I249.5
      "I249.6" { ExternalVisible := 'False'} : Bool := FALSE;   // I249.6
      "I249.7" { ExternalVisible := 'False'} : Bool := FALSE;   // I249.7
      "I250.0" { ExternalVisible := 'False'} : Bool := FALSE;   // I250.0
      "I250.1" { ExternalVisible := 'False'} : Bool := FALSE;   // I250.1
      "I250.2" { ExternalVisible := 'False'} : Bool := FALSE;   // I250.2
      "I250.3" { ExternalVisible := 'False'} : Bool := FALSE;   // I250.3
      "I250.4" { ExternalVisible := 'False'} : Bool := FALSE;   // I250.4
      "I250.5" { ExternalVisible := 'False'} : Bool := FALSE;   // I250.5
      "I250.6" { ExternalVisible := 'False'} : Bool := FALSE;   // I250.6
      "I250.7" { ExternalVisible := 'False'} : Bool := FALSE;   // I250.7
      "I251.0" { ExternalVisible := 'False'} : Bool := FALSE;   // I251.0
      "I251.1" { ExternalVisible := 'False'} : Bool := FALSE;   // I251.1
      "I251.2" { ExternalVisible := 'False'} : Bool := FALSE;   // I251.2
      "I251.3" { ExternalVisible := 'False'} : Bool := FALSE;   // I251.3
      "I251.4" { ExternalVisible := 'False'} : Bool := FALSE;   // I251.4
      "I251.5" { ExternalVisible := 'False'} : Bool := FALSE;   // I251.5
      "I251.6" { ExternalVisible := 'False'} : Bool := FALSE;   // I251.6
      "I251.7" { ExternalVisible := 'False'} : Bool := FALSE;   // I251.7
      "I252.0" { ExternalVisible := 'False'} : Bool := FALSE;   // I252.0
      "I252.1" { ExternalVisible := 'False'} : Bool := FALSE;   // I252.1
      "I252.2" { ExternalVisible := 'False'} : Bool := FALSE;   // I252.2
      "I252.3" { ExternalVisible := 'False'} : Bool := FALSE;   // I252.3
      "I252.4" { ExternalVisible := 'False'} : Bool := FALSE;   // I252.4
      "I252.5" { ExternalVisible := 'False'} : Bool := FALSE;   // I252.5
      "I252.6" { ExternalVisible := 'False'} : Bool := FALSE;   // I252.6
      "I252.7" { ExternalVisible := 'False'} : Bool := FALSE;   // I252.7
      "I253.0" { ExternalVisible := 'False'} : Bool := FALSE;   // I253.0
      "I253.1" { ExternalVisible := 'False'} : Bool := FALSE;   // I253.1
      "I253.2" { ExternalVisible := 'False'} : Bool := FALSE;   // I253.2
      "I253.3" { ExternalVisible := 'False'} : Bool := FALSE;   // I253.3
      "I253.4" { ExternalVisible := 'False'} : Bool := FALSE;   // I253.4
      "I253.5" { ExternalVisible := 'False'} : Bool := FALSE;   // I253.5
      "I253.6" { ExternalVisible := 'False'} : Bool := FALSE;   // I253.6
      "I253.7" { ExternalVisible := 'False'} : Bool := FALSE;   // I253.7
      "I254.0" { ExternalVisible := 'False'} : Bool := FALSE;   // I254.0
      "I254.1" { ExternalVisible := 'False'} : Bool := FALSE;   // I254.1
      "I254.2" { ExternalVisible := 'False'} : Bool := FALSE;   // I254.2
      "I254.3" { ExternalVisible := 'False'} : Bool := FALSE;   // I254.3
      "I254.4" { ExternalVisible := 'False'} : Bool := FALSE;   // I254.4
      "I254.5" { ExternalVisible := 'False'} : Bool := FALSE;   // I254.5
      "I254.6" { ExternalVisible := 'False'} : Bool := FALSE;   // I254.6
      "I254.7" { ExternalVisible := 'False'} : Bool := FALSE;   // I254.7
      "I255.0" { ExternalVisible := 'False'} : Bool := FALSE;   // I255.0
      "I255.1" { ExternalVisible := 'False'} : Bool := FALSE;   // I255.1
      "I255.2" { ExternalVisible := 'False'} : Bool := FALSE;   // I255.2
      "I255.3" { ExternalVisible := 'False'} : Bool := FALSE;   // I255.3
      "I255.4" { ExternalVisible := 'False'} : Bool := FALSE;   // I255.4
      "I255.5" { ExternalVisible := 'False'} : Bool := FALSE;   // I255.5
      "I255.6" { ExternalVisible := 'False'} : Bool := FALSE;   // I255.6
      "I255.7" { ExternalVisible := 'False'} : Bool := FALSE;   // I255.7
      "I256.0" { ExternalVisible := 'False'} : Bool := FALSE;   // I256.0
      "I256.1" { ExternalVisible := 'False'} : Bool := FALSE;   // I256.1
      "I256.2" { ExternalVisible := 'False'} : Bool := FALSE;   // I256.2
      "I256.3" { ExternalVisible := 'False'} : Bool := FALSE;   // I256.3
      "I256.4" { ExternalVisible := 'False'} : Bool := FALSE;   // I256.4
      "I256.5" { ExternalVisible := 'False'} : Bool := FALSE;   // I256.5
      "I256.6" { ExternalVisible := 'False'} : Bool := FALSE;   // I256.6
      "I256.7" { ExternalVisible := 'False'} : Bool := FALSE;   // I256.7
      "I257.0" { ExternalVisible := 'False'} : Bool := FALSE;   // I257.0
      "I257.1" { ExternalVisible := 'False'} : Bool := FALSE;   // I257.1
      "I257.2" { ExternalVisible := 'False'} : Bool := FALSE;   // I257.2
      "I257.3" { ExternalVisible := 'False'} : Bool := FALSE;   // I257.3
      "I257.4" { ExternalVisible := 'False'} : Bool := FALSE;   // I257.4
      "I257.5" { ExternalVisible := 'False'} : Bool := FALSE;   // I257.5
      "I257.6" { ExternalVisible := 'False'} : Bool := FALSE;   // I257.6
      "I257.7" { ExternalVisible := 'False'} : Bool := FALSE;   // I257.7
      "I258.0" { ExternalVisible := 'False'} : Bool := FALSE;   // I258.0
      "I258.1" { ExternalVisible := 'False'} : Bool := FALSE;   // I258.1
      "I258.2" { ExternalVisible := 'False'} : Bool := FALSE;   // I258.2
      "I258.3" { ExternalVisible := 'False'} : Bool := FALSE;   // I258.3
      "I258.4" { ExternalVisible := 'False'} : Bool := FALSE;   // I258.4
      "I258.5" { ExternalVisible := 'False'} : Bool := FALSE;   // I258.5
      "I258.6" { ExternalVisible := 'False'} : Bool := FALSE;   // I258.6
      "I258.7" { ExternalVisible := 'False'} : Bool := FALSE;   // I258.7
      "I259.0" { ExternalVisible := 'False'} : Bool := FALSE;   // I259.0
      "I259.1" { ExternalVisible := 'False'} : Bool := FALSE;   // I259.1
      "I259.2" { ExternalVisible := 'False'} : Bool := FALSE;   // I259.2
      "I259.3" { ExternalVisible := 'False'} : Bool := FALSE;   // I259.3
      "I259.4" { ExternalVisible := 'False'} : Bool := FALSE;   // I259.4
      "I259.5" { ExternalVisible := 'False'} : Bool := FALSE;   // I259.5
      "I259.6" { ExternalVisible := 'False'} : Bool := FALSE;   // I259.6
      "I259.7" { ExternalVisible := 'False'} : Bool := FALSE;   // I259.7
      "I260.0" { ExternalVisible := 'False'} : Bool := FALSE;   // I260.0
      "I260.1" { ExternalVisible := 'False'} : Bool := FALSE;   // I260.1
      "I260.2" { ExternalVisible := 'False'} : Bool := FALSE;   // I260.2
      "I260.3" { ExternalVisible := 'False'} : Bool := FALSE;   // I260.3
      "I260.4" { ExternalVisible := 'False'} : Bool := FALSE;   // I260.4
      "I260.5" { ExternalVisible := 'False'} : Bool := FALSE;   // I260.5
      "I260.6" { ExternalVisible := 'False'} : Bool := FALSE;   // I260.6
      "I260.7" { ExternalVisible := 'False'} : Bool := FALSE;   // I260.7
      "I261.0" { ExternalVisible := 'False'} : Bool := FALSE;   // I261.0
      "I261.1" { ExternalVisible := 'False'} : Bool := FALSE;   // I261.1
      "I261.2" { ExternalVisible := 'False'} : Bool := FALSE;   // I261.2
      "I261.3" { ExternalVisible := 'False'} : Bool := FALSE;   // I261.3
      "I261.4" { ExternalVisible := 'False'} : Bool := FALSE;   // I261.4
      "I261.5" { ExternalVisible := 'False'} : Bool := FALSE;   // I261.5
      "I261.6" { ExternalVisible := 'False'} : Bool := FALSE;   // I261.6
      "I261.7" { ExternalVisible := 'False'} : Bool := FALSE;   // I261.7
      "I262.0" { ExternalVisible := 'False'} : Bool := FALSE;   // I262.0
      "I262.1" { ExternalVisible := 'False'} : Bool := FALSE;   // I262.1
      "I262.2" { ExternalVisible := 'False'} : Bool := FALSE;   // I262.2
      "I262.3" { ExternalVisible := 'False'} : Bool := FALSE;   // I262.3
      "I262.4" { ExternalVisible := 'False'} : Bool := FALSE;   // I262.4
      "I262.5" { ExternalVisible := 'False'} : Bool := FALSE;   // I262.5
      "I262.6" { ExternalVisible := 'False'} : Bool := FALSE;   // I262.6
      "I262.7" { ExternalVisible := 'False'} : Bool := FALSE;   // I262.7
      "I263.0" { ExternalVisible := 'False'} : Bool := FALSE;   // I263.0
      "I263.1" { ExternalVisible := 'False'} : Bool := FALSE;   // I263.1
      "I263.2" { ExternalVisible := 'False'} : Bool := FALSE;   // I263.2
      "I263.3" { ExternalVisible := 'False'} : Bool := FALSE;   // I263.3
      "I263.4" { ExternalVisible := 'False'} : Bool := FALSE;   // I263.4
      "I263.5" { ExternalVisible := 'False'} : Bool := FALSE;   // I263.5
      "I263.6" { ExternalVisible := 'False'} : Bool := FALSE;   // I263.6
      "I263.7" { ExternalVisible := 'False'} : Bool := FALSE;   // I263.7
      "I264.0" { ExternalVisible := 'False'} : Bool := FALSE;   // I264.0
      "I264.1" { ExternalVisible := 'False'} : Bool := FALSE;   // I264.1
      "I264.2" { ExternalVisible := 'False'} : Bool := FALSE;   // I264.2
      "I264.3" { ExternalVisible := 'False'} : Bool := FALSE;   // I264.3
      "I264.4" { ExternalVisible := 'False'} : Bool := FALSE;   // I264.4
      "I264.5" { ExternalVisible := 'False'} : Bool := FALSE;   // I264.5
      "I264.6" { ExternalVisible := 'False'} : Bool := FALSE;   // I264.6
      "I264.7" { ExternalVisible := 'False'} : Bool := FALSE;   // I264.7
      "I265.0" { ExternalVisible := 'False'} : Bool := FALSE;   // I265.0
      "I265.1" { ExternalVisible := 'False'} : Bool := FALSE;   // I265.1
      "I265.2" { ExternalVisible := 'False'} : Bool := FALSE;   // I265.2
      "I265.3" { ExternalVisible := 'False'} : Bool := FALSE;   // I265.3
      "I265.4" { ExternalVisible := 'False'} : Bool := FALSE;   // I265.4
      "I265.5" { ExternalVisible := 'False'} : Bool := FALSE;   // I265.5
      "I265.6" { ExternalVisible := 'False'} : Bool := FALSE;   // I265.6
      "I265.7" { ExternalVisible := 'False'} : Bool := FALSE;   // I265.7
      "I266.0" { ExternalVisible := 'False'} : Bool := FALSE;   // I266.0
      "I266.1" { ExternalVisible := 'False'} : Bool := FALSE;   // I266.1
      "I266.2" { ExternalVisible := 'False'} : Bool := FALSE;   // I266.2
      "I266.3" { ExternalVisible := 'False'} : Bool := FALSE;   // I266.3
      "I266.4" { ExternalVisible := 'False'} : Bool := FALSE;   // I266.4
      "I266.5" { ExternalVisible := 'False'} : Bool := FALSE;   // I266.5
      "I266.6" { ExternalVisible := 'False'} : Bool := FALSE;   // I266.6
      "I266.7" { ExternalVisible := 'False'} : Bool := FALSE;   // I266.7
      "I267.0" { ExternalVisible := 'False'} : Bool := FALSE;   // I267.0
      "I267.1" { ExternalVisible := 'False'} : Bool := FALSE;   // I267.1
      "I267.2" { ExternalVisible := 'False'} : Bool := FALSE;   // I267.2
      "I267.3" { ExternalVisible := 'False'} : Bool := FALSE;   // I267.3
      "I267.4" { ExternalVisible := 'False'} : Bool := FALSE;   // I267.4
      "I267.5" { ExternalVisible := 'False'} : Bool := FALSE;   // I267.5
      "I267.6" { ExternalVisible := 'False'} : Bool := FALSE;   // I267.6
      "I267.7" { ExternalVisible := 'False'} : Bool := FALSE;   // I267.7
      "I268.0" { ExternalVisible := 'False'} : Bool := FALSE;   // I268.0
      "I268.1" { ExternalVisible := 'False'} : Bool := FALSE;   // I268.1
      "I268.2" { ExternalVisible := 'False'} : Bool := FALSE;   // I268.2
      "I268.3" { ExternalVisible := 'False'} : Bool := FALSE;   // I268.3
      "I268.4" { ExternalVisible := 'False'} : Bool := FALSE;   // I268.4
      "I268.5" { ExternalVisible := 'False'} : Bool := FALSE;   // I268.5
      "I268.6" { ExternalVisible := 'False'} : Bool := FALSE;   // I268.6
      "I268.7" { ExternalVisible := 'False'} : Bool := FALSE;   // I268.7
      "I269.0" { ExternalVisible := 'False'} : Bool := FALSE;   // I269.0
      "I269.1" { ExternalVisible := 'False'} : Bool := FALSE;   // I269.1
      "I269.2" { ExternalVisible := 'False'} : Bool := FALSE;   // I269.2
      "I269.3" { ExternalVisible := 'False'} : Bool := FALSE;   // I269.3
      "I269.4" { ExternalVisible := 'False'} : Bool := FALSE;   // I269.4
      "I269.5" { ExternalVisible := 'False'} : Bool := FALSE;   // I269.5
      "I269.6" { ExternalVisible := 'False'} : Bool := FALSE;   // I269.6
      "I269.7" { ExternalVisible := 'False'} : Bool := FALSE;   // I269.7
      "I270.0" { ExternalVisible := 'False'} : Bool := FALSE;   // I270.0
      "I270.1" { ExternalVisible := 'False'} : Bool := FALSE;   // I270.1
      "I270.2" { ExternalVisible := 'False'} : Bool := FALSE;   // I270.2
      "I270.3" { ExternalVisible := 'False'} : Bool := FALSE;   // I270.3
      "I270.4" { ExternalVisible := 'False'} : Bool := FALSE;   // I270.4
      "I270.5" { ExternalVisible := 'False'} : Bool := FALSE;   // I270.5
      "I270.6" { ExternalVisible := 'False'} : Bool := FALSE;   // I270.6
      "I270.7" { ExternalVisible := 'False'} : Bool := FALSE;   // I270.7
      "I271.0" { ExternalVisible := 'False'} : Bool := FALSE;   // I271.0
      "I271.1" { ExternalVisible := 'False'} : Bool := FALSE;   // I271.1
      "I271.2" { ExternalVisible := 'False'} : Bool := FALSE;   // I271.2
      "I271.3" { ExternalVisible := 'False'} : Bool := FALSE;   // I271.3
      "I271.4" { ExternalVisible := 'False'} : Bool := FALSE;   // I271.4
      "I271.5" { ExternalVisible := 'False'} : Bool := FALSE;   // I271.5
      "I271.6" { ExternalVisible := 'False'} : Bool := FALSE;   // I271.6
      "I271.7" { ExternalVisible := 'False'} : Bool := FALSE;   // I271.7
      "I272.0" { ExternalVisible := 'False'} : Bool := FALSE;   // I272.0
      "I272.1" { ExternalVisible := 'False'} : Bool := FALSE;   // I272.1
      "I272.2" { ExternalVisible := 'False'} : Bool := FALSE;   // I272.2
      "I272.3" { ExternalVisible := 'False'} : Bool := FALSE;   // I272.3
      "I272.4" { ExternalVisible := 'False'} : Bool := FALSE;   // I272.4
      "I272.5" { ExternalVisible := 'False'} : Bool := FALSE;   // I272.5
      "I272.6" { ExternalVisible := 'False'} : Bool := FALSE;   // I272.6
      "I272.7" { ExternalVisible := 'False'} : Bool := FALSE;   // I272.7
      "I273.0" { ExternalVisible := 'False'} : Bool := FALSE;   // I273.0
      "I273.1" { ExternalVisible := 'False'} : Bool := FALSE;   // I273.1
      "I273.2" { ExternalVisible := 'False'} : Bool := FALSE;   // I273.2
      "I273.3" { ExternalVisible := 'False'} : Bool := FALSE;   // I273.3
      "I273.4" { ExternalVisible := 'False'} : Bool := FALSE;   // I273.4
      "I273.5" { ExternalVisible := 'False'} : Bool := FALSE;   // I273.5
      "I273.6" { ExternalVisible := 'False'} : Bool := FALSE;   // I273.6
      "I273.7" { ExternalVisible := 'False'} : Bool := FALSE;   // I273.7
      "I274.0" { ExternalVisible := 'False'} : Bool := FALSE;   // I274.0
      "I274.1" { ExternalVisible := 'False'} : Bool := FALSE;   // I274.1
      "I274.2" { ExternalVisible := 'False'} : Bool := FALSE;   // I274.2
      "I274.3" { ExternalVisible := 'False'} : Bool := FALSE;   // I274.3
      "I274.4" { ExternalVisible := 'False'} : Bool := FALSE;   // I274.4
      "I274.5" { ExternalVisible := 'False'} : Bool := FALSE;   // I274.5
      "I274.6" { ExternalVisible := 'False'} : Bool := FALSE;   // I274.6
      "I274.7" { ExternalVisible := 'False'} : Bool := FALSE;   // I274.7
      "I275.0" { ExternalVisible := 'False'} : Bool := FALSE;   // I275.0
      "I275.1" { ExternalVisible := 'False'} : Bool := FALSE;   // I275.1
      "I275.2" { ExternalVisible := 'False'} : Bool := FALSE;   // I275.2
      "I275.3" { ExternalVisible := 'False'} : Bool := FALSE;   // I275.3
      "I275.4" { ExternalVisible := 'False'} : Bool := FALSE;   // I275.4
      "I275.5" { ExternalVisible := 'False'} : Bool := FALSE;   // I275.5
      "I275.6" { ExternalVisible := 'False'} : Bool := FALSE;   // I275.6
      "I275.7" { ExternalVisible := 'False'} : Bool := FALSE;   // I275.7
      "I276.0" { ExternalVisible := 'False'} : Bool := FALSE;   // I276.0
      "I276.1" { ExternalVisible := 'False'} : Bool := FALSE;   // I276.1
      "I276.2" { ExternalVisible := 'False'} : Bool := FALSE;   // I276.2
      "I276.3" { ExternalVisible := 'False'} : Bool := FALSE;   // I276.3
      "I276.4" { ExternalVisible := 'False'} : Bool := FALSE;   // I276.4
      "I276.5" { ExternalVisible := 'False'} : Bool := FALSE;   // I276.5
      "I276.6" { ExternalVisible := 'False'} : Bool := FALSE;   // I276.6
      "I276.7" { ExternalVisible := 'False'} : Bool := FALSE;   // I276.7
      "I277.0" { ExternalVisible := 'False'} : Bool := FALSE;   // I277.0
      "I277.1" { ExternalVisible := 'False'} : Bool := FALSE;   // I277.1
      "I277.2" { ExternalVisible := 'False'} : Bool := FALSE;   // I277.2
      "I277.3" { ExternalVisible := 'False'} : Bool := FALSE;   // I277.3
      "I277.4" { ExternalVisible := 'False'} : Bool := FALSE;   // I277.4
      "I277.5" { ExternalVisible := 'False'} : Bool := FALSE;   // I277.5
      "I277.6" { ExternalVisible := 'False'} : Bool := FALSE;   // I277.6
      "I277.7" { ExternalVisible := 'False'} : Bool := FALSE;   // I277.7
      "I278.0" { ExternalVisible := 'False'} : Bool := FALSE;   // I278.0
      "I278.1" { ExternalVisible := 'False'} : Bool := FALSE;   // I278.1
      "I278.2" { ExternalVisible := 'False'} : Bool := FALSE;   // I278.2
      "I278.3" { ExternalVisible := 'False'} : Bool := FALSE;   // I278.3
      "I278.4" { ExternalVisible := 'False'} : Bool := FALSE;   // I278.4
      "I278.5" { ExternalVisible := 'False'} : Bool := FALSE;   // I278.5
      "I278.6" { ExternalVisible := 'False'} : Bool := FALSE;   // I278.6
      "I278.7" { ExternalVisible := 'False'} : Bool := FALSE;   // I278.7
      "I279.0" { ExternalVisible := 'False'} : Bool := FALSE;   // I279.0
      "I279.1" { ExternalVisible := 'False'} : Bool := FALSE;   // I279.1
      "I279.2" { ExternalVisible := 'False'} : Bool := FALSE;   // I279.2
      "I279.3" { ExternalVisible := 'False'} : Bool := FALSE;   // I279.3
      "I279.4" { ExternalVisible := 'False'} : Bool := FALSE;   // I279.4
      "I279.5" { ExternalVisible := 'False'} : Bool := FALSE;   // I279.5
      "I279.6" { ExternalVisible := 'False'} : Bool := FALSE;   // I279.6
      "I279.7" { ExternalVisible := 'False'} : Bool := FALSE;   // I279.7
      "I280.0" { ExternalVisible := 'False'} : Bool := FALSE;   // I280.0
      "I280.1" { ExternalVisible := 'False'} : Bool := FALSE;   // I280.1
      "I280.2" { ExternalVisible := 'False'} : Bool := FALSE;   // I280.2
      "I280.3" { ExternalVisible := 'False'} : Bool := FALSE;   // I280.3
      "I280.4" { ExternalVisible := 'False'} : Bool := FALSE;   // I280.4
      "I280.5" { ExternalVisible := 'False'} : Bool := FALSE;   // I280.5
      "I280.6" { ExternalVisible := 'False'} : Bool := FALSE;   // I280.6
      "I280.7" { ExternalVisible := 'False'} : Bool := FALSE;   // I280.7
      "I281.0" { ExternalVisible := 'False'} : Bool := FALSE;   // I281.0
      "I281.1" { ExternalVisible := 'False'} : Bool := FALSE;   // I281.1
      "I281.2" { ExternalVisible := 'False'} : Bool := FALSE;   // I281.2
      "I281.3" { ExternalVisible := 'False'} : Bool := FALSE;   // I281.3
      "I281.4" { ExternalVisible := 'False'} : Bool := FALSE;   // I281.4
      "I281.5" { ExternalVisible := 'False'} : Bool := FALSE;   // I281.5
      "I281.6" { ExternalVisible := 'False'} : Bool := FALSE;   // I281.6
      "I281.7" { ExternalVisible := 'False'} : Bool := FALSE;   // I281.7
      "I282.0" { ExternalVisible := 'False'} : Bool := FALSE;   // I282.0
      "I282.1" { ExternalVisible := 'False'} : Bool := FALSE;   // I282.1
      "I282.2" { ExternalVisible := 'False'} : Bool := FALSE;   // I282.2
      "I282.3" { ExternalVisible := 'False'} : Bool := FALSE;   // I282.3
      "I282.4" { ExternalVisible := 'False'} : Bool := FALSE;   // I282.4
      "I282.5" { ExternalVisible := 'False'} : Bool := FALSE;   // I282.5
      "I282.6" { ExternalVisible := 'False'} : Bool := FALSE;   // I282.6
      "I282.7" { ExternalVisible := 'False'} : Bool := FALSE;   // I282.7
      "I283.0" { ExternalVisible := 'False'} : Bool := FALSE;   // I283.0
      "I283.1" { ExternalVisible := 'False'} : Bool := FALSE;   // I283.1
      "I283.2" { ExternalVisible := 'False'} : Bool := FALSE;   // I283.2
      "I283.3" { ExternalVisible := 'False'} : Bool := FALSE;   // I283.3
      "I283.4" { ExternalVisible := 'False'} : Bool := FALSE;   // I283.4
      "I283.5" { ExternalVisible := 'False'} : Bool := FALSE;   // I283.5
      "I283.6" { ExternalVisible := 'False'} : Bool := FALSE;   // I283.6
      "I283.7" { ExternalVisible := 'False'} : Bool := FALSE;   // I283.7
      "I284.0" { ExternalVisible := 'False'} : Bool := FALSE;   // I284.0
      "I284.1" { ExternalVisible := 'False'} : Bool := FALSE;   // I284.1
      "I284.2" { ExternalVisible := 'False'} : Bool := FALSE;   // I284.2
      "I284.3" { ExternalVisible := 'False'} : Bool := FALSE;   // I284.3
      "I284.4" { ExternalVisible := 'False'} : Bool := FALSE;   // I284.4
      "I284.5" { ExternalVisible := 'False'} : Bool := FALSE;   // I284.5
      "I284.6" { ExternalVisible := 'False'} : Bool := FALSE;   // I284.6
      "I284.7" { ExternalVisible := 'False'} : Bool := FALSE;   // I284.7
      "I285.0" { ExternalVisible := 'False'} : Bool := FALSE;   // I285.0
      "I285.1" { ExternalVisible := 'False'} : Bool := FALSE;   // I285.1
      "I285.2" { ExternalVisible := 'False'} : Bool := FALSE;   // I285.2
      "I285.3" { ExternalVisible := 'False'} : Bool := FALSE;   // I285.3
      "I285.4" { ExternalVisible := 'False'} : Bool := FALSE;   // I285.4
      "I285.5" { ExternalVisible := 'False'} : Bool := FALSE;   // I285.5
      "I285.6" { ExternalVisible := 'False'} : Bool := FALSE;   // I285.6
      "I285.7" { ExternalVisible := 'False'} : Bool := FALSE;   // I285.7
      "I286.0" { ExternalVisible := 'False'} : Bool := FALSE;   // I286.0
      "I286.1" { ExternalVisible := 'False'} : Bool := FALSE;   // I286.1
      "I286.2" { ExternalVisible := 'False'} : Bool := FALSE;   // I286.2
      "I286.3" { ExternalVisible := 'False'} : Bool := FALSE;   // I286.3
      "I286.4" { ExternalVisible := 'False'} : Bool := FALSE;   // I286.4
      "I286.5" { ExternalVisible := 'False'} : Bool := FALSE;   // I286.5
      "I286.6" { ExternalVisible := 'False'} : Bool := FALSE;   // I286.6
      "I286.7" { ExternalVisible := 'False'} : Bool := FALSE;   // I286.7
      "I287.0" { ExternalVisible := 'False'} : Bool := FALSE;   // I287.0
      "I287.1" { ExternalVisible := 'False'} : Bool := FALSE;   // I287.1
      "I287.2" { ExternalVisible := 'False'} : Bool := FALSE;   // I287.2
      "I287.3" { ExternalVisible := 'False'} : Bool := FALSE;   // I287.3
      "I287.4" { ExternalVisible := 'False'} : Bool := FALSE;   // I287.4
      "I287.5" { ExternalVisible := 'False'} : Bool := FALSE;   // I287.5
      "I287.6" { ExternalVisible := 'False'} : Bool := FALSE;   // I287.6
      "I287.7" { ExternalVisible := 'False'} : Bool := FALSE;   // I287.7
      "I288.0" { ExternalVisible := 'False'} : Bool := FALSE;   // I288.0
      "I288.1" { ExternalVisible := 'False'} : Bool := FALSE;   // I288.1
      "I288.2" { ExternalVisible := 'False'} : Bool := FALSE;   // I288.2
      "I288.3" { ExternalVisible := 'False'} : Bool := FALSE;   // I288.3
      "I288.4" { ExternalVisible := 'False'} : Bool := FALSE;   // I288.4
      "I288.5" { ExternalVisible := 'False'} : Bool := FALSE;   // I288.5
      "I288.6" { ExternalVisible := 'False'} : Bool := FALSE;   // I288.6
      "I288.7" { ExternalVisible := 'False'} : Bool := FALSE;   // I288.7
      "I289.0" { ExternalVisible := 'False'} : Bool := FALSE;   // I289.0
      "I289.1" { ExternalVisible := 'False'} : Bool := FALSE;   // I289.1
      "I289.2" { ExternalVisible := 'False'} : Bool := FALSE;   // I289.2
      "I289.3" { ExternalVisible := 'False'} : Bool := FALSE;   // I289.3
      "I289.4" { ExternalVisible := 'False'} : Bool := FALSE;   // I289.4
      "I289.5" { ExternalVisible := 'False'} : Bool := FALSE;   // I289.5
      "I289.6" { ExternalVisible := 'False'} : Bool := FALSE;   // I289.6
      "I289.7" { ExternalVisible := 'False'} : Bool := FALSE;   // I289.7
      "I290.0" { ExternalVisible := 'False'} : Bool := FALSE;   // I290.0
      "I290.1" { ExternalVisible := 'False'} : Bool := FALSE;   // I290.1
      "I290.2" { ExternalVisible := 'False'} : Bool := FALSE;   // I290.2
      "I290.3" { ExternalVisible := 'False'} : Bool := FALSE;   // I290.3
      "I290.4" { ExternalVisible := 'False'} : Bool := FALSE;   // I290.4
      "I290.5" { ExternalVisible := 'False'} : Bool := FALSE;   // I290.5
      "I290.6" { ExternalVisible := 'False'} : Bool := FALSE;   // I290.6
      "I290.7" { ExternalVisible := 'False'} : Bool := FALSE;   // I290.7
      "I291.0" { ExternalVisible := 'False'} : Bool := FALSE;   // I291.0
      "I291.1" { ExternalVisible := 'False'} : Bool := FALSE;   // I291.1
      "I291.2" { ExternalVisible := 'False'} : Bool := FALSE;   // I291.2
      "I291.3" { ExternalVisible := 'False'} : Bool := FALSE;   // I291.3
      "I291.4" { ExternalVisible := 'False'} : Bool := FALSE;   // I291.4
      "I291.5" { ExternalVisible := 'False'} : Bool := FALSE;   // I291.5
      "I291.6" { ExternalVisible := 'False'} : Bool := FALSE;   // I291.6
      "I291.7" { ExternalVisible := 'False'} : Bool := FALSE;   // I291.7
      "I292.0" { ExternalVisible := 'False'} : Bool := FALSE;   // I292.0
      "I292.1" { ExternalVisible := 'False'} : Bool := FALSE;   // I292.1
      "I292.2" { ExternalVisible := 'False'} : Bool := FALSE;   // I292.2
      "I292.3" { ExternalVisible := 'False'} : Bool := FALSE;   // I292.3
      "I292.4" { ExternalVisible := 'False'} : Bool := FALSE;   // I292.4
      "I292.5" { ExternalVisible := 'False'} : Bool := FALSE;   // I292.5
      "I292.6" { ExternalVisible := 'False'} : Bool := FALSE;   // I292.6
      "I292.7" { ExternalVisible := 'False'} : Bool := FALSE;   // I292.7
      "I293.0" { ExternalVisible := 'False'} : Bool := FALSE;   // I293.0
      "I293.1" { ExternalVisible := 'False'} : Bool := FALSE;   // I293.1
      "I293.2" { ExternalVisible := 'False'} : Bool := FALSE;   // I293.2
      "I293.3" { ExternalVisible := 'False'} : Bool := FALSE;   // I293.3
      "I293.4" { ExternalVisible := 'False'} : Bool := FALSE;   // I293.4
      "I293.5" { ExternalVisible := 'False'} : Bool := FALSE;   // I293.5
      "I293.6" { ExternalVisible := 'False'} : Bool := FALSE;   // I293.6
      "I293.7" { ExternalVisible := 'False'} : Bool := FALSE;   // I293.7
      "I294.0" { ExternalVisible := 'False'} : Bool := FALSE;   // I294.0
      "I294.1" { ExternalVisible := 'False'} : Bool := FALSE;   // I294.1
      "I294.2" { ExternalVisible := 'False'} : Bool := FALSE;   // I294.2
      "I294.3" { ExternalVisible := 'False'} : Bool := FALSE;   // I294.3
      "I294.4" { ExternalVisible := 'False'} : Bool := FALSE;   // I294.4
      "I294.5" { ExternalVisible := 'False'} : Bool := FALSE;   // I294.5
      "I294.6" { ExternalVisible := 'False'} : Bool := FALSE;   // I294.6
      "I294.7" { ExternalVisible := 'False'} : Bool := FALSE;   // I294.7
      "I295.0" { ExternalVisible := 'False'} : Bool := FALSE;   // I295.0
      "I295.1" { ExternalVisible := 'False'} : Bool := FALSE;   // I295.1
      "I295.2" { ExternalVisible := 'False'} : Bool := FALSE;   // I295.2
      "I295.3" { ExternalVisible := 'False'} : Bool := FALSE;   // I295.3
      "I295.4" { ExternalVisible := 'False'} : Bool := FALSE;   // I295.4
      "I295.5" { ExternalVisible := 'False'} : Bool := FALSE;   // I295.5
      "I295.6" { ExternalVisible := 'False'} : Bool := FALSE;   // I295.6
      "I295.7" { ExternalVisible := 'False'} : Bool := FALSE;   // I295.7
      "I296.0" { ExternalVisible := 'False'} : Bool := FALSE;   // I296.0
      "I296.1" { ExternalVisible := 'False'} : Bool := FALSE;   // I296.1
      "I296.2" { ExternalVisible := 'False'} : Bool := FALSE;   // I296.2
      "I296.3" { ExternalVisible := 'False'} : Bool := FALSE;   // I296.3
      "I296.4" { ExternalVisible := 'False'} : Bool := FALSE;   // I296.4
      "I296.5" { ExternalVisible := 'False'} : Bool := FALSE;   // I296.5
      "I296.6" { ExternalVisible := 'False'} : Bool := FALSE;   // I296.6
      "I296.7" { ExternalVisible := 'False'} : Bool := FALSE;   // I296.7
      "I297.0" { ExternalVisible := 'False'} : Bool := FALSE;   // I297.0
      "I297.1" { ExternalVisible := 'False'} : Bool := FALSE;   // I297.1
      "I297.2" { ExternalVisible := 'False'} : Bool := FALSE;   // I297.2
      "I297.3" { ExternalVisible := 'False'} : Bool := FALSE;   // I297.3
      "I297.4" { ExternalVisible := 'False'} : Bool := FALSE;   // I297.4
      "I297.5" { ExternalVisible := 'False'} : Bool := FALSE;   // I297.5
      "I297.6" { ExternalVisible := 'False'} : Bool := FALSE;   // I297.6
      "I297.7" { ExternalVisible := 'False'} : Bool := FALSE;   // I297.7
      "I298.0" { ExternalVisible := 'False'} : Bool := FALSE;   // I298.0
      "I298.1" { ExternalVisible := 'False'} : Bool := FALSE;   // I298.1
      "I298.2" { ExternalVisible := 'False'} : Bool := FALSE;   // I298.2
      "I298.3" { ExternalVisible := 'False'} : Bool := FALSE;   // I298.3
      "I298.4" { ExternalVisible := 'False'} : Bool := FALSE;   // I298.4
      "I298.5" { ExternalVisible := 'False'} : Bool := FALSE;   // I298.5
      "I298.6" { ExternalVisible := 'False'} : Bool := FALSE;   // I298.6
      "I298.7" { ExternalVisible := 'False'} : Bool := FALSE;   // I298.7
      "I299.0" { ExternalVisible := 'False'} : Bool := FALSE;   // I299.0
      "I299.1" { ExternalVisible := 'False'} : Bool := FALSE;   // I299.1
      "I299.2" { ExternalVisible := 'False'} : Bool := FALSE;   // I299.2
      "I299.3" { ExternalVisible := 'False'} : Bool := FALSE;   // I299.3
      "I299.4" { ExternalVisible := 'False'} : Bool := FALSE;   // I299.4
      "I299.5" { ExternalVisible := 'False'} : Bool := FALSE;   // I299.5
      "I299.6" { ExternalVisible := 'False'} : Bool := FALSE;   // I299.6
      "I299.7" { ExternalVisible := 'False'} : Bool := FALSE;   // I299.7
      "I300.0" { ExternalVisible := 'False'} : Bool := FALSE;   // I300.0
      "I300.1" { ExternalVisible := 'False'} : Bool := FALSE;   // I300.1
      "I300.2" { ExternalVisible := 'False'} : Bool := FALSE;   // I300.2
      "I300.3" { ExternalVisible := 'False'} : Bool := FALSE;   // I300.3
      "I300.4" { ExternalVisible := 'False'} : Bool := FALSE;   // I300.4
      "I300.5" { ExternalVisible := 'False'} : Bool := FALSE;   // I300.5
      "I300.6" { ExternalVisible := 'False'} : Bool := FALSE;   // I300.6
      "I300.7" { ExternalVisible := 'False'} : Bool := FALSE;   // I300.7
      "I301.0" { ExternalVisible := 'False'} : Bool := FALSE;   // I301.0
      "I301.1" { ExternalVisible := 'False'} : Bool := FALSE;   // I301.1
      "I301.2" { ExternalVisible := 'False'} : Bool := FALSE;   // I301.2
      "I301.3" { ExternalVisible := 'False'} : Bool := FALSE;   // I301.3
      "I301.4" { ExternalVisible := 'False'} : Bool := FALSE;   // I301.4
      "I301.5" { ExternalVisible := 'False'} : Bool := FALSE;   // I301.5
      "I301.6" { ExternalVisible := 'False'} : Bool := FALSE;   // I301.6
      "I301.7" { ExternalVisible := 'False'} : Bool := FALSE;   // I301.7
      "I302.0" { ExternalVisible := 'False'} : Bool := FALSE;   // I302.0
      "I302.1" { ExternalVisible := 'False'} : Bool := FALSE;   // I302.1
      "I302.2" { ExternalVisible := 'False'} : Bool := FALSE;   // I302.2
      "I302.3" { ExternalVisible := 'False'} : Bool := FALSE;   // I302.3
      "I302.4" { ExternalVisible := 'False'} : Bool := FALSE;   // I302.4
      "I302.5" { ExternalVisible := 'False'} : Bool := FALSE;   // I302.5
      "I302.6" { ExternalVisible := 'False'} : Bool := FALSE;   // I302.6
      "I302.7" { ExternalVisible := 'False'} : Bool := FALSE;   // I302.7
      "I303.0" { ExternalVisible := 'False'} : Bool := FALSE;   // I303.0
      "I303.1" { ExternalVisible := 'False'} : Bool := FALSE;   // I303.1
      "I303.2" { ExternalVisible := 'False'} : Bool := FALSE;   // I303.2
      "I303.3" { ExternalVisible := 'False'} : Bool := FALSE;   // I303.3
      "I303.4" { ExternalVisible := 'False'} : Bool := FALSE;   // I303.4
      "I303.5" { ExternalVisible := 'False'} : Bool := FALSE;   // I303.5
      "I303.6" { ExternalVisible := 'False'} : Bool := FALSE;   // I303.6
      "I303.7" { ExternalVisible := 'False'} : Bool := FALSE;   // I303.7
      "I304.0" { ExternalVisible := 'False'} : Bool := FALSE;   // I304.0
      "I304.1" { ExternalVisible := 'False'} : Bool := FALSE;   // I304.1
      "I304.2" { ExternalVisible := 'False'} : Bool := FALSE;   // I304.2
      "I304.3" { ExternalVisible := 'False'} : Bool := FALSE;   // I304.3
      "I304.4" { ExternalVisible := 'False'} : Bool := FALSE;   // I304.4
      "I304.5" { ExternalVisible := 'False'} : Bool := FALSE;   // I304.5
      "I304.6" { ExternalVisible := 'False'} : Bool := FALSE;   // I304.6
      "I304.7" { ExternalVisible := 'False'} : Bool := FALSE;   // I304.7
      "I305.0" { ExternalVisible := 'False'} : Bool := FALSE;   // I305.0
      "I305.1" { ExternalVisible := 'False'} : Bool := FALSE;   // I305.1
      "I305.2" { ExternalVisible := 'False'} : Bool := FALSE;   // I305.2
      "I305.3" { ExternalVisible := 'False'} : Bool := FALSE;   // I305.3
      "I305.4" { ExternalVisible := 'False'} : Bool := FALSE;   // I305.4
      "I305.5" { ExternalVisible := 'False'} : Bool := FALSE;   // I305.5
      "I305.6" { ExternalVisible := 'False'} : Bool := FALSE;   // I305.6
      "I305.7" { ExternalVisible := 'False'} : Bool := FALSE;   // I305.7
      "I306.0" { ExternalVisible := 'False'} : Bool := FALSE;   // I306.0
      "I306.1" { ExternalVisible := 'False'} : Bool := FALSE;   // I306.1
      "I306.2" { ExternalVisible := 'False'} : Bool := FALSE;   // I306.2
      "I306.3" { ExternalVisible := 'False'} : Bool := FALSE;   // I306.3
      "I306.4" { ExternalVisible := 'False'} : Bool := FALSE;   // I306.4
      "I306.5" { ExternalVisible := 'False'} : Bool := FALSE;   // I306.5
      "I306.6" { ExternalVisible := 'False'} : Bool := FALSE;   // I306.6
      "I306.7" { ExternalVisible := 'False'} : Bool := FALSE;   // I306.7
      "I307.0" { ExternalVisible := 'False'} : Bool := FALSE;   // I307.0
      "I307.1" { ExternalVisible := 'False'} : Bool := FALSE;   // I307.1
      "I307.2" { ExternalVisible := 'False'} : Bool := FALSE;   // I307.2
      "I307.3" { ExternalVisible := 'False'} : Bool := FALSE;   // I307.3
      "I307.4" { ExternalVisible := 'False'} : Bool := FALSE;   // I307.4
      "I307.5" { ExternalVisible := 'False'} : Bool := FALSE;   // I307.5
      "I307.6" { ExternalVisible := 'False'} : Bool := FALSE;   // I307.6
      "I307.7" { ExternalVisible := 'False'} : Bool := FALSE;   // I307.7
      "I308.0" { ExternalVisible := 'False'} : Bool := FALSE;   // I308.0
      "I308.1" { ExternalVisible := 'False'} : Bool := FALSE;   // I308.1
      "I308.2" { ExternalVisible := 'False'} : Bool := FALSE;   // I308.2
      "I308.3" { ExternalVisible := 'False'} : Bool := FALSE;   // I308.3
      "I308.4" { ExternalVisible := 'False'} : Bool := FALSE;   // I308.4
      "I308.5" { ExternalVisible := 'False'} : Bool := FALSE;   // I308.5
      "I308.6" { ExternalVisible := 'False'} : Bool := FALSE;   // I308.6
      "I308.7" { ExternalVisible := 'False'} : Bool := FALSE;   // I308.7
      "I309.0" { ExternalVisible := 'False'} : Bool := FALSE;   // I309.0
      "I309.1" { ExternalVisible := 'False'} : Bool := FALSE;   // I309.1
      "I309.2" { ExternalVisible := 'False'} : Bool := FALSE;   // I309.2
      "I309.3" { ExternalVisible := 'False'} : Bool := FALSE;   // I309.3
      "I309.4" { ExternalVisible := 'False'} : Bool := FALSE;   // I309.4
      "I309.5" { ExternalVisible := 'False'} : Bool := FALSE;   // I309.5
      "I309.6" { ExternalVisible := 'False'} : Bool := FALSE;   // I309.6
      "I309.7" { ExternalVisible := 'False'} : Bool := FALSE;   // I309.7
      "I310.0" { ExternalVisible := 'False'} : Bool := FALSE;   // I310.0
      "I310.1" { ExternalVisible := 'False'} : Bool := FALSE;   // I310.1
      "I310.2" { ExternalVisible := 'False'} : Bool := FALSE;   // I310.2
      "I310.3" { ExternalVisible := 'False'} : Bool := FALSE;   // I310.3
      "I310.4" { ExternalVisible := 'False'} : Bool := FALSE;   // I310.4
      "I310.5" { ExternalVisible := 'False'} : Bool := FALSE;   // I310.5
      "I310.6" { ExternalVisible := 'False'} : Bool := FALSE;   // I310.6
      "I310.7" { ExternalVisible := 'False'} : Bool := FALSE;   // I310.7
      "I311.0" { ExternalVisible := 'False'} : Bool := FALSE;   // I311.0
      "I311.1" { ExternalVisible := 'False'} : Bool := FALSE;   // I311.1
      "I311.2" { ExternalVisible := 'False'} : Bool := FALSE;   // I311.2
      "I311.3" { ExternalVisible := 'False'} : Bool := FALSE;   // I311.3
      "I311.4" { ExternalVisible := 'False'} : Bool := FALSE;   // I311.4
      "I311.5" { ExternalVisible := 'False'} : Bool := FALSE;   // I311.5
      "I311.6" { ExternalVisible := 'False'} : Bool := FALSE;   // I311.6
      "I311.7" { ExternalVisible := 'False'} : Bool := FALSE;   // I311.7
      "I312.0" { ExternalVisible := 'False'} : Bool := FALSE;   // I312.0
      "I312.1" { ExternalVisible := 'False'} : Bool := FALSE;   // I312.1
      "I312.2" { ExternalVisible := 'False'} : Bool := FALSE;   // I312.2
      "I312.3" { ExternalVisible := 'False'} : Bool := FALSE;   // I312.3
      "I312.4" { ExternalVisible := 'False'} : Bool := FALSE;   // I312.4
      "I312.5" { ExternalVisible := 'False'} : Bool := FALSE;   // I312.5
      "I312.6" { ExternalVisible := 'False'} : Bool := FALSE;   // I312.6
      "I312.7" { ExternalVisible := 'False'} : Bool := FALSE;   // I312.7
      "I313.0" { ExternalVisible := 'False'} : Bool := FALSE;   // I313.0
      "I313.1" { ExternalVisible := 'False'} : Bool := FALSE;   // I313.1
      "I313.2" { ExternalVisible := 'False'} : Bool := FALSE;   // I313.2
      "I313.3" { ExternalVisible := 'False'} : Bool := FALSE;   // I313.3
      "I313.4" { ExternalVisible := 'False'} : Bool := FALSE;   // I313.4
      "I313.5" { ExternalVisible := 'False'} : Bool := FALSE;   // I313.5
      "I313.6" { ExternalVisible := 'False'} : Bool := FALSE;   // I313.6
      "I313.7" { ExternalVisible := 'False'} : Bool := FALSE;   // I313.7
      "I314.0" { ExternalVisible := 'False'} : Bool := FALSE;   // I314.0
      "I314.1" { ExternalVisible := 'False'} : Bool := FALSE;   // I314.1
      "I314.2" { ExternalVisible := 'False'} : Bool := FALSE;   // I314.2
      "I314.3" { ExternalVisible := 'False'} : Bool := FALSE;   // I314.3
      "I314.4" { ExternalVisible := 'False'} : Bool := FALSE;   // I314.4
      "I314.5" { ExternalVisible := 'False'} : Bool := FALSE;   // I314.5
      "I314.6" { ExternalVisible := 'False'} : Bool := FALSE;   // I314.6
      "I314.7" { ExternalVisible := 'False'} : Bool := FALSE;   // I314.7
      "I315.0" { ExternalVisible := 'False'} : Bool := FALSE;   // I315.0
      "I315.1" { ExternalVisible := 'False'} : Bool := FALSE;   // I315.1
      "I315.2" { ExternalVisible := 'False'} : Bool := FALSE;   // I315.2
      "I315.3" { ExternalVisible := 'False'} : Bool := FALSE;   // I315.3
      "I315.4" { ExternalVisible := 'False'} : Bool := FALSE;   // I315.4
      "I315.5" { ExternalVisible := 'False'} : Bool := FALSE;   // I315.5
      "I315.6" { ExternalVisible := 'False'} : Bool := FALSE;   // I315.6
      "I315.7" { ExternalVisible := 'False'} : Bool := FALSE;   // I315.7
      "I316.0" { ExternalVisible := 'False'} : Bool := FALSE;   // I316.0
      "I316.1" { ExternalVisible := 'False'} : Bool := FALSE;   // I316.1
      "I316.2" { ExternalVisible := 'False'} : Bool := FALSE;   // I316.2
      "I316.3" { ExternalVisible := 'False'} : Bool := FALSE;   // I316.3
      "I316.4" { ExternalVisible := 'False'} : Bool := FALSE;   // I316.4
      "I316.5" { ExternalVisible := 'False'} : Bool := FALSE;   // I316.5
      "I316.6" { ExternalVisible := 'False'} : Bool := FALSE;   // I316.6
      "I316.7" { ExternalVisible := 'False'} : Bool := FALSE;   // I316.7
      "I317.0" { ExternalVisible := 'False'} : Bool := FALSE;   // I317.0
      "I317.1" { ExternalVisible := 'False'} : Bool := FALSE;   // I317.1
      "I317.2" { ExternalVisible := 'False'} : Bool := FALSE;   // I317.2
      "I317.3" { ExternalVisible := 'False'} : Bool := FALSE;   // I317.3
      "I317.4" { ExternalVisible := 'False'} : Bool := FALSE;   // I317.4
      "I317.5" { ExternalVisible := 'False'} : Bool := FALSE;   // I317.5
      "I317.6" { ExternalVisible := 'False'} : Bool := FALSE;   // I317.6
      "I317.7" { ExternalVisible := 'False'} : Bool := FALSE;   // I317.7
      "I318.0" { ExternalVisible := 'False'} : Bool := FALSE;   // I318.0
      "I318.1" { ExternalVisible := 'False'} : Bool := FALSE;   // I318.1
      "I318.2" { ExternalVisible := 'False'} : Bool := FALSE;   // I318.2
      "I318.3" { ExternalVisible := 'False'} : Bool := FALSE;   // I318.3
      "I318.4" { ExternalVisible := 'False'} : Bool := FALSE;   // I318.4
      "I318.5" { ExternalVisible := 'False'} : Bool := FALSE;   // I318.5
      "I318.6" { ExternalVisible := 'False'} : Bool := FALSE;   // I318.6
      "I318.7" { ExternalVisible := 'False'} : Bool := FALSE;   // I318.7
      "I319.0" { ExternalVisible := 'False'} : Bool := FALSE;   // I319.0
      "I319.1" { ExternalVisible := 'False'} : Bool := FALSE;   // I319.1
      "I319.2" { ExternalVisible := 'False'} : Bool := FALSE;   // I319.2
      "I319.3" { ExternalVisible := 'False'} : Bool := FALSE;   // I319.3
      "I319.4" { ExternalVisible := 'False'} : Bool := FALSE;   // I319.4
      "I319.5" { ExternalVisible := 'False'} : Bool := FALSE;   // I319.5
      "I319.6" { ExternalVisible := 'False'} : Bool := FALSE;   // I319.6
      "I319.7" { ExternalVisible := 'False'} : Bool := FALSE;   // I319.7
      "I320.0" { ExternalVisible := 'False'} : Bool := FALSE;   // I320.0
      "I320.1" { ExternalVisible := 'False'} : Bool := FALSE;   // I320.1
      "I320.2" { ExternalVisible := 'False'} : Bool := FALSE;   // I320.2
      "I320.3" { ExternalVisible := 'False'} : Bool := FALSE;   // I320.3
      "I320.4" { ExternalVisible := 'False'} : Bool := FALSE;   // I320.4
      "I320.5" { ExternalVisible := 'False'} : Bool := FALSE;   // I320.5
      "I320.6" { ExternalVisible := 'False'} : Bool := FALSE;   // I320.6
      "I320.7" { ExternalVisible := 'False'} : Bool := FALSE;   // I320.7
      "I321.0" { ExternalVisible := 'False'} : Bool := FALSE;   // I321.0
      "I321.1" { ExternalVisible := 'False'} : Bool := FALSE;   // I321.1
      "I321.2" { ExternalVisible := 'False'} : Bool := FALSE;   // I321.2
      "I321.3" { ExternalVisible := 'False'} : Bool := FALSE;   // I321.3
      "I321.4" { ExternalVisible := 'False'} : Bool := FALSE;   // I321.4
      "I321.5" { ExternalVisible := 'False'} : Bool := FALSE;   // I321.5
      "I321.6" { ExternalVisible := 'False'} : Bool := FALSE;   // I321.6
      "I321.7" { ExternalVisible := 'False'} : Bool := FALSE;   // I321.7
      "I322.0" { ExternalVisible := 'False'} : Bool := FALSE;   // I322.0
      "I322.1" { ExternalVisible := 'False'} : Bool := FALSE;   // I322.1
      "I322.2" { ExternalVisible := 'False'} : Bool := FALSE;   // I322.2
      "I322.3" { ExternalVisible := 'False'} : Bool := FALSE;   // I322.3
      "I322.4" { ExternalVisible := 'False'} : Bool := FALSE;   // I322.4
      "I322.5" { ExternalVisible := 'False'} : Bool := FALSE;   // I322.5
      "I322.6" { ExternalVisible := 'False'} : Bool := FALSE;   // I322.6
      "I322.7" { ExternalVisible := 'False'} : Bool := FALSE;   // I322.7
      "I323.0" { ExternalVisible := 'False'} : Bool := FALSE;   // I323.0
      "I323.1" { ExternalVisible := 'False'} : Bool := FALSE;   // I323.1
      "I323.2" { ExternalVisible := 'False'} : Bool := FALSE;   // I323.2
      "I323.3" { ExternalVisible := 'False'} : Bool := FALSE;   // I323.3
      "I323.4" { ExternalVisible := 'False'} : Bool := FALSE;   // I323.4
      "I323.5" { ExternalVisible := 'False'} : Bool := FALSE;   // I323.5
      "I323.6" { ExternalVisible := 'False'} : Bool := FALSE;   // I323.6
      "I323.7" { ExternalVisible := 'False'} : Bool := FALSE;   // I323.7
      "I324.0" { ExternalVisible := 'False'} : Bool := FALSE;   // I324.0
      "I324.1" { ExternalVisible := 'False'} : Bool := FALSE;   // I324.1
      "I324.2" { ExternalVisible := 'False'} : Bool := FALSE;   // I324.2
      "I324.3" { ExternalVisible := 'False'} : Bool := FALSE;   // I324.3
      "I324.4" { ExternalVisible := 'False'} : Bool := FALSE;   // I324.4
      "I324.5" { ExternalVisible := 'False'} : Bool := FALSE;   // I324.5
      "I324.6" { ExternalVisible := 'False'} : Bool := FALSE;   // I324.6
      "I324.7" { ExternalVisible := 'False'} : Bool := FALSE;   // I324.7
      "I325.0" { ExternalVisible := 'False'} : Bool := FALSE;   // I325.0
      "I325.1" { ExternalVisible := 'False'} : Bool := FALSE;   // I325.1
      "I325.2" { ExternalVisible := 'False'} : Bool := FALSE;   // I325.2
      "I325.3" { ExternalVisible := 'False'} : Bool := FALSE;   // I325.3
      "I325.4" { ExternalVisible := 'False'} : Bool := FALSE;   // I325.4
      "I325.5" { ExternalVisible := 'False'} : Bool := FALSE;   // I325.5
      "I325.6" { ExternalVisible := 'False'} : Bool := FALSE;   // I325.6
      "I325.7" { ExternalVisible := 'False'} : Bool := FALSE;   // I325.7
      "I326.0" { ExternalVisible := 'False'} : Bool := FALSE;   // I326.0
      "I326.1" { ExternalVisible := 'False'} : Bool := FALSE;   // I326.1
      "I326.2" { ExternalVisible := 'False'} : Bool := FALSE;   // I326.2
      "I326.3" { ExternalVisible := 'False'} : Bool := FALSE;   // I326.3
      "I326.4" { ExternalVisible := 'False'} : Bool := FALSE;   // I326.4
      "I326.5" { ExternalVisible := 'False'} : Bool := FALSE;   // I326.5
      "I326.6" { ExternalVisible := 'False'} : Bool := FALSE;   // I326.6
      "I326.7" { ExternalVisible := 'False'} : Bool := FALSE;   // I326.7
      "I327.0" { ExternalVisible := 'False'} : Bool := FALSE;   // I327.0
      "I327.1" { ExternalVisible := 'False'} : Bool := FALSE;   // I327.1
      "I327.2" { ExternalVisible := 'False'} : Bool := FALSE;   // I327.2
      "I327.3" { ExternalVisible := 'False'} : Bool := FALSE;   // I327.3
      "I327.4" { ExternalVisible := 'False'} : Bool := FALSE;   // I327.4
      "I327.5" { ExternalVisible := 'False'} : Bool := FALSE;   // I327.5
      "I327.6" { ExternalVisible := 'False'} : Bool := FALSE;   // I327.6
      "I327.7" { ExternalVisible := 'False'} : Bool := FALSE;   // I327.7
      "I328.0" { ExternalVisible := 'False'} : Bool := FALSE;   // I328.0
      "I328.1" { ExternalVisible := 'False'} : Bool := FALSE;   // I328.1
      "I328.2" { ExternalVisible := 'False'} : Bool := FALSE;   // I328.2
      "I328.3" { ExternalVisible := 'False'} : Bool := FALSE;   // I328.3
      "I328.4" { ExternalVisible := 'False'} : Bool := FALSE;   // I328.4
      "I328.5" { ExternalVisible := 'False'} : Bool := FALSE;   // I328.5
      "I328.6" { ExternalVisible := 'False'} : Bool := FALSE;   // I328.6
      "I328.7" { ExternalVisible := 'False'} : Bool := FALSE;   // I328.7
      "I329.0" { ExternalVisible := 'False'} : Bool := FALSE;   // I329.0
      "I329.1" { ExternalVisible := 'False'} : Bool := FALSE;   // I329.1
      "I329.2" { ExternalVisible := 'False'} : Bool := FALSE;   // I329.2
      "I329.3" { ExternalVisible := 'False'} : Bool := FALSE;   // I329.3
      "I329.4" { ExternalVisible := 'False'} : Bool := FALSE;   // I329.4
      "I329.5" { ExternalVisible := 'False'} : Bool := FALSE;   // I329.5
      "I329.6" { ExternalVisible := 'False'} : Bool := FALSE;   // I329.6
      "I329.7" { ExternalVisible := 'False'} : Bool := FALSE;   // I329.7
      "I330.0" { ExternalVisible := 'False'} : Bool := FALSE;   // I330.0
      "I330.1" { ExternalVisible := 'False'} : Bool := FALSE;   // I330.1
      "I330.2" { ExternalVisible := 'False'} : Bool := FALSE;   // I330.2
      "I330.3" { ExternalVisible := 'False'} : Bool := FALSE;   // I330.3
      "I330.4" { ExternalVisible := 'False'} : Bool := FALSE;   // I330.4
      "I330.5" { ExternalVisible := 'False'} : Bool := FALSE;   // I330.5
      "I330.6" { ExternalVisible := 'False'} : Bool := FALSE;   // I330.6
      "I330.7" { ExternalVisible := 'False'} : Bool := FALSE;   // I330.7
      "I331.0" { ExternalVisible := 'False'} : Bool := FALSE;   // I331.0
      "I331.1" { ExternalVisible := 'False'} : Bool := FALSE;   // I331.1
      "I331.2" { ExternalVisible := 'False'} : Bool := FALSE;   // I331.2
      "I331.3" { ExternalVisible := 'False'} : Bool := FALSE;   // I331.3
      "I331.4" { ExternalVisible := 'False'} : Bool := FALSE;   // I331.4
      "I331.5" { ExternalVisible := 'False'} : Bool := FALSE;   // I331.5
      "I331.6" { ExternalVisible := 'False'} : Bool := FALSE;   // I331.6
      "I331.7" { ExternalVisible := 'False'} : Bool := FALSE;   // I331.7
      "I332.0" { ExternalVisible := 'False'} : Bool := FALSE;   // I332.0
      "I332.1" { ExternalVisible := 'False'} : Bool := FALSE;   // I332.1
      "I332.2" { ExternalVisible := 'False'} : Bool := FALSE;   // I332.2
      "I332.3" { ExternalVisible := 'False'} : Bool := FALSE;   // I332.3
      "I332.4" { ExternalVisible := 'False'} : Bool := FALSE;   // I332.4
      "I332.5" { ExternalVisible := 'False'} : Bool := FALSE;   // I332.5
      "I332.6" { ExternalVisible := 'False'} : Bool := FALSE;   // I332.6
      "I332.7" { ExternalVisible := 'False'} : Bool := FALSE;   // I332.7
      "I333.0" { ExternalVisible := 'False'} : Bool := FALSE;   // I333.0
      "I333.1" { ExternalVisible := 'False'} : Bool := FALSE;   // I333.1
      "I333.2" { ExternalVisible := 'False'} : Bool := FALSE;   // I333.2
      "I333.3" { ExternalVisible := 'False'} : Bool := FALSE;   // I333.3
      "I333.4" { ExternalVisible := 'False'} : Bool := FALSE;   // I333.4
      "I333.5" { ExternalVisible := 'False'} : Bool := FALSE;   // I333.5
      "I333.6" { ExternalVisible := 'False'} : Bool := FALSE;   // I333.6
      "I333.7" { ExternalVisible := 'False'} : Bool := FALSE;   // I333.7
      "I334.0" { ExternalVisible := 'False'} : Bool := FALSE;   // I334.0
      "I334.1" { ExternalVisible := 'False'} : Bool := FALSE;   // I334.1
      "I334.2" { ExternalVisible := 'False'} : Bool := FALSE;   // I334.2
      "I334.3" { ExternalVisible := 'False'} : Bool := FALSE;   // I334.3
      "I334.4" { ExternalVisible := 'False'} : Bool := FALSE;   // I334.4
      "I334.5" { ExternalVisible := 'False'} : Bool := FALSE;   // I334.5
      "I334.6" { ExternalVisible := 'False'} : Bool := FALSE;   // I334.6
      "I334.7" { ExternalVisible := 'False'} : Bool := FALSE;   // I334.7
      "I335.0" { ExternalVisible := 'False'} : Bool := FALSE;   // I335.0
      "I335.1" { ExternalVisible := 'False'} : Bool := FALSE;   // I335.1
      "I335.2" { ExternalVisible := 'False'} : Bool := FALSE;   // I335.2
      "I335.3" { ExternalVisible := 'False'} : Bool := FALSE;   // I335.3
      "I335.4" { ExternalVisible := 'False'} : Bool := FALSE;   // I335.4
      "I335.5" { ExternalVisible := 'False'} : Bool := FALSE;   // I335.5
      "I335.6" { ExternalVisible := 'False'} : Bool := FALSE;   // I335.6
      "I335.7" { ExternalVisible := 'False'} : Bool := FALSE;   // I335.7
      "I336.0" { ExternalVisible := 'False'} : Bool := FALSE;   // I336.0
      "I336.1" { ExternalVisible := 'False'} : Bool := FALSE;   // I336.1
      "I336.2" { ExternalVisible := 'False'} : Bool := FALSE;   // I336.2
      "I336.3" { ExternalVisible := 'False'} : Bool := FALSE;   // I336.3
      "I336.4" { ExternalVisible := 'False'} : Bool := FALSE;   // I336.4
      "I336.5" { ExternalVisible := 'False'} : Bool := FALSE;   // I336.5
      "I336.6" { ExternalVisible := 'False'} : Bool := FALSE;   // I336.6
      "I336.7" { ExternalVisible := 'False'} : Bool := FALSE;   // I336.7
      "I337.0" { ExternalVisible := 'False'} : Bool := FALSE;   // I337.0
      "I337.1" { ExternalVisible := 'False'} : Bool := FALSE;   // I337.1
      "I337.2" { ExternalVisible := 'False'} : Bool := FALSE;   // I337.2
      "I337.3" { ExternalVisible := 'False'} : Bool := FALSE;   // I337.3
      "I337.4" { ExternalVisible := 'False'} : Bool := FALSE;   // I337.4
      "I337.5" { ExternalVisible := 'False'} : Bool := FALSE;   // I337.5
      "I337.6" { ExternalVisible := 'False'} : Bool := FALSE;   // I337.6
      "I337.7" { ExternalVisible := 'False'} : Bool := FALSE;   // I337.7
      "I338.0" { ExternalVisible := 'False'} : Bool := FALSE;   // I338.0
      "I338.1" { ExternalVisible := 'False'} : Bool := FALSE;   // I338.1
      "I338.2" { ExternalVisible := 'False'} : Bool := FALSE;   // I338.2
      "I338.3" { ExternalVisible := 'False'} : Bool := FALSE;   // I338.3
      "I338.4" { ExternalVisible := 'False'} : Bool := FALSE;   // I338.4
      "I338.5" { ExternalVisible := 'False'} : Bool := FALSE;   // I338.5
      "I338.6" { ExternalVisible := 'False'} : Bool := FALSE;   // I338.6
      "I338.7" { ExternalVisible := 'False'} : Bool := FALSE;   // I338.7
      "I339.0" { ExternalVisible := 'False'} : Bool := FALSE;   // I339.0
      "I339.1" { ExternalVisible := 'False'} : Bool := FALSE;   // I339.1
      "I339.2" { ExternalVisible := 'False'} : Bool := FALSE;   // I339.2
      "I339.3" { ExternalVisible := 'False'} : Bool := FALSE;   // I339.3
      "I339.4" { ExternalVisible := 'False'} : Bool := FALSE;   // I339.4
      "I339.5" { ExternalVisible := 'False'} : Bool := FALSE;   // I339.5
      "I339.6" { ExternalVisible := 'False'} : Bool := FALSE;   // I339.6
      "I339.7" { ExternalVisible := 'False'} : Bool := FALSE;   // I339.7
      "I340.0" { ExternalVisible := 'False'} : Bool := FALSE;   // I340.0
      "I340.1" { ExternalVisible := 'False'} : Bool := FALSE;   // I340.1
      "I340.2" { ExternalVisible := 'False'} : Bool := FALSE;   // I340.2
